LIN {X 0,Y 383.746,Z 842.553,A -85,B 0,C 180,E1 14810.521,E2 14810.521} C_VEL
LIN {X 0,Y 388.275,Z 838.57,A -85,B 0,C 180,E1 14810.091,E2 14810.091} C_VEL
LIN {X 0,Y 383.695,Z 874.566,A -85,B 0,C 180,E1 14809.08,E2 14809.08} C_VEL
LIN {X 0,Y 381.946,Z 882.091,A -85,B 0,C 180,E1 14808.965,E2 14808.965} C_VEL
LIN {X 0,Y 374.562,Z 902.014,A -85,B 0,C 180,E1 14808.987,E2 14808.987} C_VEL
LIN {X 0,Y 373.141,Z 908.472,A -85,B 0,C 180,E1 14808.863,E2 14808.863} C_VEL
LIN {X 0,Y 363.178,Z 988.067,A -85,B 0,C 180,E1 14806.33,E2 14806.33} C_VEL
LIN {X 0,Y 360.037,Z 1012.069,A -85,B 0,C 180,E1 14805.364,E2 14805.364} C_VEL
LIN {X 0,Y 356.378,Z 1034.28,A -85,B 0,C 180,E1 14804.205,E2 14804.205} C_VEL
LIN {X 0,Y 351.773,Z 1057.589,A -85,B 0,C 180,E1 14802.682,E2 14802.682} C_VEL
LIN {X 0,Y 346.903,Z 1079.031,A -85,B 0,C 180,E1 14800.957,E2 14800.957} C_VEL
LIN {X 0,Y 341.537,Z 1100.164,A -85,B 0,C 180,E1 14798.901,E2 14798.901} C_VEL
LIN {X 0,Y 335.908,Z 1120.268,A -85,B 0,C 180,E1 14796.537,E2 14796.537} C_VEL
LIN {X 0,Y 330.579,Z 1138.155,A -85,B 0,C 180,E1 14794.026,E2 14794.026} C_VEL
LIN {X 0,Y 325.16,Z 1155.707,A -85,B 0,C 180,E1 14791.105,E2 14791.105} C_VEL
LIN {X 0,Y 320.4,Z 1170.927,A -85,B 0,C 180,E1 14788.115,E2 14788.115} C_VEL
LIN {X 0,Y 315.886,Z 1185.531,A -85,B 0,C 180,E1 14784.698,E2 14784.698} C_VEL
LIN {X 0,Y 312.205,Z 1197.976,A -85,B 0,C 180,E1 14781.217,E2 14781.217} C_VEL
LIN {X 0,Y 309.066,Z 1209.644,A -85,B 0,C 180,E1 14777.316,E2 14777.316} C_VEL
LIN {X 0,Y 306.838,Z 1219.359,A -85,B 0,C 180,E1 14773.378,E2 14773.378} C_VEL
LIN {X 0,Y 305.434,Z 1227.199,A -85,B 0,C 180,E1 14769.421,E2 14769.421} C_VEL
LIN {X 0,Y 304.675,Z 1233.378,A -85,B 0,C 180,E1 14765.461,E2 14765.461} C_VEL
LIN {X 0,Y 304.399,Z 1238.104,A -85,B 0,C 180,E1 14761.506,E2 14761.506} C_VEL
LIN {X 0,Y 304.384,Z 1241.144,A -85,B 0,C 180,E1 14757.741,E2 14757.741} C_VEL
LIN {X 0,Y 304.604,Z 1243.124,A -85,B 0,C 180,E1 14753.781,E2 14753.781} C_VEL
LIN {X 0,Y 305.158,Z 1243.715,A -85,B 0,C 180,E1 14749.808,E2 14749.808} C_VEL
LIN {X 0,Y 306.521,Z 1242.868,A -85,B 0,C 180,E1 14745.26,E2 14745.26} C_VEL
LIN {X 0,Y 309.14,Z 1240.272,A -85,B 0,C 180,E1 14740.54,E2 14740.54} C_VEL
LIN {X 0,Y 313.102,Z 1236.128,A -85,B 0,C 180,E1 14736.073,E2 14736.073} C_VEL
LIN {X 0,Y 318.886,Z 1230.051,A -85,B 0,C 180,E1 14731.536,E2 14731.536} C_VEL
LIN {X 0,Y 326.471,Z 1222.117,A -85,B 0,C 180,E1 14727.173,E2 14727.173} C_VEL
LIN {X 0,Y 335.463,Z 1212.699,A -85,B 0,C 180,E1 14723.194,E2 14723.194} C_VEL
LIN {X 0,Y 346.318,Z 1201.267,A -85,B 0,C 180,E1 14719.408,E2 14719.408} C_VEL
LIN {X 0,Y 359.067,Z 1187.767,A -85,B 0,C 180,E1 14715.879,E2 14715.879} C_VEL
LIN {X 0,Y 366.745,Z 1179.688,A -85,B 0,C 180,E1 14714.081,E2 14714.081} C_VEL
LIN {X 0,Y 351.897,Z 1193.932,A -85,B 0,C 180,E1 14711.242,E2 14711.242} C_VEL
LIN {X 0,Y 336.916,Z 1211.003,A -85,B 0,C 180,E1 14707.262,E2 14707.262} C_VEL
LIN {X 0,Y 323.989,Z 1229.125,A -85,B 0,C 180,E1 14702.262,E2 14702.262} C_VEL
LIN {X 0,Y 315.462,Z 1243.813,A -85,B 0,C 180,E1 14697.363,E2 14697.363} C_VEL
LIN {X 0,Y 310.275,Z 1254.664,A -85,B 0,C 180,E1 14692.953,E2 14692.953} C_VEL
LIN {X 0,Y 306.948,Z 1263.193,A -85,B 0,C 180,E1 14688.619,E2 14688.619} C_VEL
LIN {X 0,Y 305.097,Z 1269.475,A -85,B 0,C 180,E1 14684.425,E2 14684.425} C_VEL
LIN {X 0,Y 304.326,Z 1273.688,A -85,B 0,C 180,E1 14680.413,E2 14680.413} C_VEL
LIN {X 0,Y 304.222,Z 1276.03,A -85,B 0,C 180,E1 14676.608,E2 14676.608} C_VEL
LIN {X 0,Y 304.399,Z 1276.705,A -85,B 0,C 180,E1 14673.015,E2 14673.015} C_VEL
LIN {X 0,Y 304.56,Z 1275.912,A -85,B 0,C 180,E1 14669.626,E2 14669.626} C_VEL
LIN {X 0,Y 304.568,Z 1273.68,A -85,B 0,C 180,E1 14666.238,E2 14666.238} C_VEL
LIN {X 0,Y 304.521,Z 1269.98,A -85,B 0,C 180,E1 14662.835,E2 14662.835} C_VEL
LIN {X 0,Y 304.622,Z 1264.454,A -85,B 0,C 180,E1 14659.219,E2 14659.219} C_VEL
LIN {X 0,Y 305.152,Z 1256.818,A -85,B 0,C 180,E1 14655.389,E2 14655.389} C_VEL
LIN {X 0,Y 306.321,Z 1247.288,A -85,B 0,C 180,E1 14651.544,E2 14651.544} C_VEL
LIN {X 0,Y 308.437,Z 1235.038,A -85,B 0,C 180,E1 14647.512,E2 14647.512} C_VEL
LIN {X 0,Y 311.408,Z 1221.22,A -85,B 0,C 180,E1 14643.701,E2 14643.701} C_VEL
LIN {X 0,Y 315.633,Z 1204.223,A -85,B 0,C 180,E1 14639.759,E2 14639.759} C_VEL
LIN {X 0,Y 320.988,Z 1184.662,A -85,B 0,C 180,E1 14635.956,E2 14635.956} C_VEL
LIN {X 0,Y 327.072,Z 1163.735,A -85,B 0,C 180,E1 14632.533,E2 14632.533} C_VEL
LIN {X 0,Y 333.784,Z 1141.453,A -85,B 0,C 180,E1 14629.458,E2 14629.458} C_VEL
LIN {X 0,Y 340.841,Z 1118.152,A -85,B 0,C 180,E1 14626.745,E2 14626.745} C_VEL
LIN {X 0,Y 348.53,Z 1092.821,A -85,B 0,C 180,E1 14624.258,E2 14624.258} C_VEL
LIN {X 0,Y 356.345,Z 1066.796,A -85,B 0,C 180,E1 14622.116,E2 14622.116} C_VEL
LIN {X 0,Y 363.648,Z 1041.389,A -85,B 0,C 180,E1 14620.395,E2 14620.395} C_VEL
LIN {X 0,Y 371.162,Z 1013.758,A -85,B 0,C 180,E1 14618.876,E2 14618.876} C_VEL
LIN {X 0,Y 377.143,Z 988.406,A -85,B 0,C 180,E1 14617.706,E2 14617.706} C_VEL
LIN {X 0,Y 371.129,Z 963.994,A -85,B 0,C 180,E1 14615.41,E2 14615.41} C_VEL
LIN {X 0,Y 366.924,Z 941.456,A -85,B 0,C 180,E1 14613.531,E2 14613.531} C_VEL
LIN {X 0,Y 363.372,Z 914.987,A -85,B 0,C 180,E1 14611.591,E2 14611.591} C_VEL
LIN {X 0,Y 361.819,Z 891.552,A -85,B 0,C 180,E1 14610.013,E2 14610.013} C_VEL
LIN {X 0,Y 372.049,Z 851.191,A -85,B 0,C 180,E1 14605.212,E2 14605.212} C_VEL
LIN {X 0,Y 380.821,Z 818.494,A -85,B 0,C 180,E1 14601.324,E2 14601.324} C_VEL
LIN {X 0,Y 381.9,Z 814.099,A -85,B 0,C 180,E1 14600.787,E2 14600.787} C_VEL
LIN {X 0,Y 375.953,Z 797.311,A -85,B 0,C 180,E1 14597.011,E2 14597.011} C_VEL
LIN {X 0,Y 370.417,Z 782.695,A -85,B 0,C 180,E1 14593.423,E2 14593.423} C_VEL
LIN {X 0,Y 364.786,Z 768.438,A -85,B 0,C 180,E1 14589.625,E2 14589.625} C_VEL
LIN {X 0,Y 359.48,Z 755.657,A -85,B 0,C 180,E1 14585.907,E2 14585.907} C_VEL
LIN {X 0,Y 354.12,Z 743.204,A -85,B 0,C 180,E1 14581.942,E2 14581.942} C_VEL
LIN {X 0,Y 349.074,Z 731.964,A -85,B 0,C 180,E1 14578.03,E2 14578.03} C_VEL
LIN {X 0,Y 344.556,Z 722.244,A -85,B 0,C 180,E1 14574.338,E2 14574.338} C_VEL
LIN {X 0,Y 340.097,Z 712.564,A -85,B 0,C 180,E1 14570.353,E2 14570.353} C_VEL
LIN {X 0,Y 336.736,Z 705.94,A -85,B 0,C 180,E1 14567.307,E2 14567.307} C_VEL
LIN {X 0,Y 334.521,Z 701.406,A -85,B 0,C 180,E1 14565.104,E2 14565.104} C_VEL
LIN {X 0,Y 332.667,Z 697.681,A -85,B 0,C 180,E1 14563.229,E2 14563.229} C_VEL
LIN {X 0,Y 330.716,Z 693.689,A -85,B 0,C 180,E1 14561.125,E2 14561.125} C_VEL
LIN {X 0,Y 328.472,Z 689.184,A -85,B 0,C 180,E1 14558.575,E2 14558.575} C_VEL
LIN {X 0,Y 326.1,Z 684.518,A -85,B 0,C 180,E1 14555.74,E2 14555.74} C_VEL
LIN {X 0,Y 323.782,Z 679.957,A -85,B 0,C 180,E1 14552.79,E2 14552.79} C_VEL
LIN {X 0,Y 321.463,Z 675.343,A -85,B 0,C 180,E1 14549.535,E2 14549.535} C_VEL
LIN {X 0,Y 323.347,Z 676.36,A -85,B 0,C 180,E1 14548.908,E2 14548.908} C_VEL
LIN {X 0,Y 329.514,Z 688.003,A -85,B 0,C 180,E1 14545.849,E2 14545.849} C_VEL
LIN {X 0,Y 335.679,Z 701.279,A -85,B 0,C 180,E1 14542.794,E2 14542.794} C_VEL
LIN {X 0,Y 341.917,Z 716.478,A -85,B 0,C 180,E1 14539.738,E2 14539.738} C_VEL
LIN {X 0,Y 347.429,Z 732.534,A -85,B 0,C 180,E1 14536.88,E2 14536.88} C_VEL
LIN {X 0,Y 352.001,Z 748.58,A -85,B 0,C 180,E1 14534.341,E2 14534.341} C_VEL
LIN {X 0,Y 346.421,Z 794.632,A -85,B 0,C 180,E1 14530.169,E2 14530.169} C_VEL
LIN {X 0,Y 340.819,Z 844.347,A -85,B 0,C 180,E1 14525.716,E2 14525.716} C_VEL
LIN {X 0,Y 338.058,Z 873.297,A -85,B 0,C 180,E1 14523.219,E2 14523.219} C_VEL
LIN {X 0,Y 338.378,Z 880.004,A -85,B 0,C 180,E1 14523.012,E2 14523.012} C_VEL
LIN {X 0,Y 332.419,Z 1032.548,A -85,B 0,C 180,E1 14519.855,E2 14519.855} C_VEL
LIN {X 0,Y 331.822,Z 1052.049,A -85,B 0,C 180,E1 14519.278,E2 14519.278} C_VEL
LIN {X 0,Y 330.671,Z 1068.771,A -85,B 0,C 180,E1 14518.487,E2 14518.487} C_VEL
LIN {X 0,Y 328.942,Z 1084.738,A -85,B 0,C 180,E1 14517.426,E2 14517.426} C_VEL
LIN {X 0,Y 326.673,Z 1100.489,A -85,B 0,C 180,E1 14516.052,E2 14516.052} C_VEL
LIN {X 0,Y 324.079,Z 1115.176,A -85,B 0,C 180,E1 14514.418,E2 14514.418} C_VEL
LIN {X 0,Y 321.235,Z 1128.864,A -85,B 0,C 180,E1 14512.508,E2 14512.508} C_VEL
LIN {X 0,Y 318.391,Z 1140.966,A -85,B 0,C 180,E1 14510.398,E2 14510.398} C_VEL
LIN {X 0,Y 315.444,Z 1152.469,A -85,B 0,C 180,E1 14507.904,E2 14507.904} C_VEL
LIN {X 0,Y 312.77,Z 1162.396,A -85,B 0,C 180,E1 14505.195,E2 14505.195} C_VEL
LIN {X 0,Y 310.464,Z 1170.688,A -85,B 0,C 180,E1 14502.27,E2 14502.27} C_VEL
LIN {X 0,Y 308.629,Z 1177.374,A -85,B 0,C 180,E1 14499.132,E2 14499.132} C_VEL
LIN {X 0,Y 307.388,Z 1182.154,A -85,B 0,C 180,E1 14495.972,E2 14495.972} C_VEL
LIN {X 0,Y 306.666,Z 1185.162,A -85,B 0,C 180,E1 14492.801,E2 14492.801} C_VEL
LIN {X 0,Y 306.392,Z 1186.519,A -85,B 0,C 180,E1 14489.437,E2 14489.437} C_VEL
LIN {X 0,Y 306.581,Z 1186.104,A -85,B 0,C 180,E1 14486.07,E2 14486.07} C_VEL
LIN {X 0,Y 307.219,Z 1184.055,A -85,B 0,C 180,E1 14482.893,E2 14482.893} C_VEL
LIN {X 0,Y 308.37,Z 1180.265,A -85,B 0,C 180,E1 14479.725,E2 14479.725} C_VEL
LIN {X 0,Y 310.095,Z 1174.632,A -85,B 0,C 180,E1 14476.573,E2 14476.573} C_VEL
LIN {X 0,Y 312.31,Z 1167.487,A -85,B 0,C 180,E1 14473.634,E2 14473.634} C_VEL
LIN {X 0,Y 314.919,Z 1158.895,A -85,B 0,C 180,E1 14470.909,E2 14470.909} C_VEL
LIN {X 0,Y 317.812,Z 1148.821,A -85,B 0,C 180,E1 14468.399,E2 14468.399} C_VEL
LIN {X 0,Y 320.876,Z 1137.312,A -85,B 0,C 180,E1 14466.101,E2 14466.101} C_VEL
LIN {X 0,Y 324.011,Z 1124.278,A -85,B 0,C 180,E1 14464.008,E2 14464.008} C_VEL
LIN {X 0,Y 326.967,Z 1110.208,A -85,B 0,C 180,E1 14462.2,E2 14462.2} C_VEL
LIN {X 0,Y 329.607,Z 1094.995,A -85,B 0,C 180,E1 14460.662,E2 14460.662} C_VEL
LIN {X 0,Y 331.831,Z 1078.659,A -85,B 0,C 180,E1 14459.385,E2 14459.385} C_VEL
LIN {X 0,Y 333.495,Z 1061.599,A -85,B 0,C 180,E1 14458.396,E2 14458.396} C_VEL
LIN {X 0,Y 334.442,Z 1044.124,A -85,B 0,C 180,E1 14457.715,E2 14457.715} C_VEL
LIN {X 0,Y 335.857,Z 997.984,A -85,B 0,C 180,E1 14456.674,E2 14456.674} C_VEL
LIN {X 0,Y 340.682,Z 888.138,A -85,B 0,C 180,E1 14454.417,E2 14454.417} C_VEL
LIN {X 0,Y 342.316,Z 888.44,A -85,B 0,C 180,E1 14454.149,E2 14454.149} C_VEL
LIN {X 0,Y 344.514,Z 886.501,A -85,B 0,C 180,E1 14453.925,E2 14453.925} C_VEL
LIN {X 0,Y 347.947,Z 880.496,A -85,B 0,C 180,E1 14453.739,E2 14453.739} C_VEL
LIN {X 0,Y 349.926,Z 876.513,A -85,B 0,C 180,E1 14453.661,E2 14453.661} C_VEL
LIN {X 0,Y 354.255,Z 874.098,A -85,B 0,C 180,E1 14453.143,E2 14453.143} C_VEL
LIN {X 0,Y 358.913,Z 869.497,A -85,B 0,C 180,E1 14452.702,E2 14452.702} C_VEL
LIN {X 0,Y 365.117,Z 865.492,A -85,B 0,C 180,E1 14452.011,E2 14452.011} C_VEL
LIN {X 0,Y 369.888,Z 861.076,A -85,B 0,C 180,E1 14451.555,E2 14451.555} C_VEL
LIN {X 0,Y 375.918,Z 856.95,A -85,B 0,C 180,E1 14450.919,E2 14450.919} C_VEL
LIN {X 0,Y 380.175,Z 853.157,A -85,B 0,C 180,E1 14450.517,E2 14450.517} C_VEL
LIN {X 0,Y 380.46,Z 853.179,A -85,B 0,C 180,E1 14450.477,E2 14450.477} C_VEL
LIN {X 0,Y 373.141,Z 908.472,A -85,B 0,C 180,E1 14448.863,E2 14448.863} C_VEL
LIN {X 0,Y 371.361,Z 915.986,A -85,B 0,C 180,E1 14448.736,E2 14448.736} C_VEL
LIN {X 0,Y 363.787,Z 935.843,A -85,B 0,C 180,E1 14448.725,E2 14448.725} C_VEL
LIN {X 0,Y 362.352,Z 942.286,A -85,B 0,C 180,E1 14448.588,E2 14448.588} C_VEL
LIN {X 0,Y 355.036,Z 1000.064,A -85,B 0,C 180,E1 14446.594,E2 14446.594} C_VEL
LIN {X 0,Y 351.627,Z 1022.777,A -85,B 0,C 180,E1 14445.541,E2 14445.541} C_VEL
LIN {X 0,Y 347.34,Z 1046.129,A -85,B 0,C 180,E1 14444.159,E2 14444.159} C_VEL
LIN {X 0,Y 342.711,Z 1067.461,A -85,B 0,C 180,E1 14442.601,E2 14442.601} C_VEL
LIN {X 0,Y 337.432,Z 1088.949,A -85,B 0,C 180,E1 14440.686,E2 14440.686} C_VEL
LIN {X 0,Y 331.833,Z 1109.386,A -85,B 0,C 180,E1 14438.48,E2 14438.48} C_VEL
LIN {X 0,Y 326.28,Z 1128.261,A -85,B 0,C 180,E1 14436.043,E2 14436.043} C_VEL
LIN {X 0,Y 320.49,Z 1146.894,A -85,B 0,C 180,E1 14433.176,E2 14433.176} C_VEL
LIN {X 0,Y 315.42,Z 1162.839,A -85,B 0,C 180,E1 14430.268,E2 14430.268} C_VEL
LIN {X 0,Y 310.338,Z 1178.724,A -85,B 0,C 180,E1 14426.81,E2 14426.81} C_VEL
LIN {X 0,Y 306.13,Z 1192.235,A -85,B 0,C 180,E1 14423.279,E2 14423.279} C_VEL
LIN {X 0,Y 302.608,Z 1204.374,A -85,B 0,C 180,E1 14419.495,E2 14419.495} C_VEL
LIN {X 0,Y 299.977,Z 1214.644,A -85,B 0,C 180,E1 14415.664,E2 14415.664} C_VEL
LIN {X 0,Y 298.104,Z 1223.506,A -85,B 0,C 180,E1 14411.61,E2 14411.61} C_VEL
LIN {X 0,Y 296.995,Z 1230.615,A -85,B 0,C 180,E1 14407.545,E2 14407.545} C_VEL
LIN {X 0,Y 296.494,Z 1236.194,A -85,B 0,C 180,E1 14403.48,E2 14403.48} C_VEL
LIN {X 0,Y 296.374,Z 1240.036,A -85,B 0,C 180,E1 14399.613,E2 14399.613} C_VEL
LIN {X 0,Y 296.488,Z 1242.863,A -85,B 0,C 180,E1 14395.357,E2 14395.357} C_VEL
LIN {X 0,Y 296.921,Z 1244.215,A -85,B 0,C 180,E1 14391.284,E2 14391.284} C_VEL
LIN {X 0,Y 297.971,Z 1244.194,A -85,B 0,C 180,E1 14386.81,E2 14386.81} C_VEL
LIN {X 0,Y 300.24,Z 1242.517,A -85,B 0,C 180,E1 14381.958,E2 14381.958} C_VEL
LIN {X 0,Y 304.013,Z 1239.12,A -85,B 0,C 180,E1 14377.164,E2 14377.164} C_VEL
LIN {X 0,Y 309.508,Z 1233.987,A -85,B 0,C 180,E1 14372.485,E2 14372.485} C_VEL
LIN {X 0,Y 316.836,Z 1227.095,A -85,B 0,C 180,E1 14367.982,E2 14367.982} C_VEL
LIN {X 0,Y 326.049,Z 1218.391,A -85,B 0,C 180,E1 14363.71,E2 14363.71} C_VEL
LIN {X 0,Y 337.135,Z 1207.821,A -85,B 0,C 180,E1 14359.717,E2 14359.717} C_VEL
LIN {X 0,Y 350.229,Z 1195.277,A -85,B 0,C 180,E1 14356.011,E2 14356.011} C_VEL
LIN {X 0,Y 357.971,Z 1187.89,A -85,B 0,C 180,E1 14354.182,E2 14354.182} C_VEL
LIN {X 0,Y 342.431,Z 1202.026,A -85,B 0,C 180,E1 14351.073,E2 14351.073} C_VEL
LIN {X 0,Y 327.659,Z 1217.995,A -85,B 0,C 180,E1 14346.956,E2 14346.956} C_VEL
LIN {X 0,Y 314.933,Z 1234.715,A -85,B 0,C 180,E1 14341.808,E2 14341.808} C_VEL
LIN {X 0,Y 306.554,Z 1248.183,A -85,B 0,C 180,E1 14336.754,E2 14336.754} C_VEL
LIN {X 0,Y 301.384,Z 1258.338,A -85,B 0,C 180,E1 14332.02,E2 14332.02} C_VEL
LIN {X 0,Y 298.359,Z 1265.813,A -85,B 0,C 180,E1 14327.557,E2 14327.557} C_VEL
LIN {X 0,Y 296.743,Z 1271.328,A -85,B 0,C 180,E1 14323.05,E2 14323.05} C_VEL
LIN {X 0,Y 296.226,Z 1274.562,A -85,B 0,C 180,E1 14318.935,E2 14318.935} C_VEL
LIN {X 0,Y 296.294,Z 1275.941,A -85,B 0,C 180,E1 14315.23,E2 14315.23} C_VEL
LIN {X 0,Y 296.515,Z 1275.809,A -85,B 0,C 180,E1 14311.548,E2 14311.548} C_VEL
LIN {X 0,Y 296.621,Z 1274.367,A -85,B 0,C 180,E1 14308.264,E2 14308.264} C_VEL
LIN {X 0,Y 296.59,Z 1271.419,A -85,B 0,C 180,E1 14304.78,E2 14304.78} C_VEL
LIN {X 0,Y 296.565,Z 1266.986,A -85,B 0,C 180,E1 14301.276,E2 14301.276} C_VEL
LIN {X 0,Y 296.821,Z 1260.651,A -85,B 0,C 180,E1 14297.552,E2 14297.552} C_VEL
LIN {X 0,Y 297.622,Z 1252.148,A -85,B 0,C 180,E1 14293.611,E2 14293.611} C_VEL
LIN {X 0,Y 299.172,Z 1241.673,A -85,B 0,C 180,E1 14289.663,E2 14289.663} C_VEL
LIN {X 0,Y 301.778,Z 1228.416,A -85,B 0,C 180,E1 14285.536,E2 14285.536} C_VEL
LIN {X 0,Y 305.101,Z 1214.292,A -85,B 0,C 180,E1 14281.834,E2 14281.834} C_VEL
LIN {X 0,Y 309.645,Z 1197.173,A -85,B 0,C 180,E1 14278.026,E2 14278.026} C_VEL
LIN {X 0,Y 315.287,Z 1177.61,A -85,B 0,C 180,E1 14274.362,E2 14274.362} C_VEL
LIN {X 0,Y 321.53,Z 1156.956,A -85,B 0,C 180,E1 14271.088,E2 14271.088} C_VEL
LIN {X 0,Y 328.465,Z 1134.516,A -85,B 0,C 180,E1 14268.077,E2 14268.077} C_VEL
LIN {X 0,Y 336.889,Z 1107.478,A -85,B 0,C 180,E1 14265.063,E2 14265.063} C_VEL
LIN {X 0,Y 344.781,Z 1082.032,A -85,B 0,C 180,E1 14262.683,E2 14262.683} C_VEL
LIN {X 0,Y 352.629,Z 1056.096,A -85,B 0,C 180,E1 14260.684,E2 14260.684} C_VEL
LIN {X 0,Y 360.592,Z 1028.573,A -85,B 0,C 180,E1 14258.945,E2 14258.945} C_VEL
LIN {X 0,Y 367.813,Z 1001.505,A -85,B 0,C 180,E1 14257.549,E2 14257.549} C_VEL
LIN {X 0,Y 370.29,Z 990.176,A -85,B 0,C 180,E1 14257.025,E2 14257.025} C_VEL
LIN {X 0,Y 364.693,Z 965.814,A -85,B 0,C 180,E1 14254.667,E2 14254.667} C_VEL
LIN {X 0,Y 360.301,Z 940.519,A -85,B 0,C 180,E1 14252.535,E2 14252.535} C_VEL
LIN {X 0,Y 357.231,Z 914.188,A -85,B 0,C 180,E1 14250.59,E2 14250.59} C_VEL
LIN {X 0,Y 355.891,Z 889.583,A -85,B 0,C 180,E1 14248.941,E2 14248.941} C_VEL
LIN {X 0,Y 365.743,Z 852.148,A -85,B 0,C 180,E1 14244.45,E2 14244.45} C_VEL
LIN {X 0,Y 374.483,Z 820.314,A -85,B 0,C 180,E1 14240.637,E2 14240.637} C_VEL
LIN {X 0,Y 375.145,Z 817.467,A -85,B 0,C 180,E1 14240.273,E2 14240.273} C_VEL
LIN {X 0,Y 369.598,Z 801.679,A -85,B 0,C 180,E1 14236.665,E2 14236.665} C_VEL
LIN {X 0,Y 364.088,Z 787.029,A -85,B 0,C 180,E1 14233.014,E2 14233.014} C_VEL
LIN {X 0,Y 358.292,Z 772.182,A -85,B 0,C 180,E1 14228.991,E2 14228.991} C_VEL
LIN {X 0,Y 352.77,Z 758.933,A -85,B 0,C 180,E1 14225.041,E2 14225.041} C_VEL
LIN {X 0,Y 347.641,Z 746.903,A -85,B 0,C 180,E1 14221.154,E2 14221.154} C_VEL
LIN {X 0,Y 342.056,Z 734.282,A -85,B 0,C 180,E1 14216.648,E2 14216.648} C_VEL
LIN {X 0,Y 336.652,Z 722.607,A -85,B 0,C 180,E1 14211.976,E2 14211.976} C_VEL
LIN {X 0,Y 332.172,Z 713.221,A -85,B 0,C 180,E1 14207.836,E2 14207.836} C_VEL
LIN {X 0,Y 328.212,Z 704.901,A -85,B 0,C 180,E1 14203.814,E2 14203.814} C_VEL
LIN {X 0,Y 325.086,Z 699.043,A -85,B 0,C 180,E1 14200.599,E2 14200.599} C_VEL
LIN {X 0,Y 323.236,Z 695.16,A -85,B 0,C 180,E1 14198.401,E2 14198.401} C_VEL
LIN {X 0,Y 320.841,Z 690.451,A -85,B 0,C 180,E1 14195.499,E2 14195.499} C_VEL
LIN {X 0,Y 318.575,Z 685.943,A -85,B 0,C 180,E1 14192.524,E2 14192.524} C_VEL
LIN {X 0,Y 316.716,Z 682.164,A -85,B 0,C 180,E1 14189.869,E2 14189.869} C_VEL
LIN {X 0,Y 319.085,Z 683.348,A -85,B 0,C 180,E1 14189.075,E2 14189.075} C_VEL
LIN {X 0,Y 324.101,Z 693.003,A -85,B 0,C 180,E1 14186.479,E2 14186.479} C_VEL
LIN {X 0,Y 330.142,Z 706.097,A -85,B 0,C 180,E1 14183.37,E2 14183.37} C_VEL
LIN {X 0,Y 336.189,Z 721.204,A -85,B 0,C 180,E1 14180.249,E2 14180.249} C_VEL
LIN {X 0,Y 341.489,Z 736.768,A -85,B 0,C 180,E1 14177.439,E2 14177.439} C_VEL
LIN {X 0,Y 345.719,Z 751.902,A -85,B 0,C 180,E1 14174.997,E2 14174.997} C_VEL
LIN {X 0,Y 339.578,Z 800.369,A -85,B 0,C 180,E1 14170.563,E2 14170.563} C_VEL
LIN {X 0,Y 333.79,Z 850.487,A -85,B 0,C 180,E1 14166.046,E2 14166.046} C_VEL
LIN {X 0,Y 331.464,Z 874.294,A -85,B 0,C 180,E1 14163.981,E2 14163.981} C_VEL
LIN {X 0,Y 331.759,Z 880.873,A -85,B 0,C 180,E1 14163.774,E2 14163.774} C_VEL
LIN {X 0,Y 325.585,Z 1032.92,A -85,B 0,C 180,E1 14160.577,E2 14160.577} C_VEL
LIN {X 0,Y 324.956,Z 1052.733,A -85,B 0,C 180,E1 14159.985,E2 14159.985} C_VEL
LIN {X 0,Y 323.721,Z 1069.933,A -85,B 0,C 180,E1 14159.157,E2 14159.157} C_VEL
LIN {X 0,Y 321.925,Z 1085.838,A -85,B 0,C 180,E1 14158.077,E2 14158.077} C_VEL
LIN {X 0,Y 319.567,Z 1101.568,A -85,B 0,C 180,E1 14156.676,E2 14156.676} C_VEL
LIN {X 0,Y 316.874,Z 1116.233,A -85,B 0,C 180,E1 14155.011,E2 14155.011} C_VEL
LIN {X 0,Y 313.921,Z 1129.897,A -85,B 0,C 180,E1 14153.062,E2 14153.062} C_VEL
LIN {X 0,Y 310.966,Z 1141.986,A -85,B 0,C 180,E1 14150.908,E2 14150.908} C_VEL
LIN {X 0,Y 307.901,Z 1153.479,A -85,B 0,C 180,E1 14148.358,E2 14148.358} C_VEL
LIN {X 0,Y 305.115,Z 1163.396,A -85,B 0,C 180,E1 14145.585,E2 14145.585} C_VEL
LIN {X 0,Y 302.708,Z 1171.676,A -85,B 0,C 180,E1 14142.589,E2 14142.589} C_VEL
LIN {X 0,Y 300.79,Z 1178.355,A -85,B 0,C 180,E1 14139.372,E2 14139.372} C_VEL
LIN {X 0,Y 299.49,Z 1183.126,A -85,B 0,C 180,E1 14136.13,E2 14136.13} C_VEL
LIN {X 0,Y 298.733,Z 1186.124,A -85,B 0,C 180,E1 14132.875,E2 14132.875} C_VEL
LIN {X 0,Y 298.448,Z 1187.473,A -85,B 0,C 180,E1 14129.422,E2 14129.422} C_VEL
LIN {X 0,Y 298.651,Z 1187.052,A -85,B 0,C 180,E1 14125.966,E2 14125.966} C_VEL
LIN {X 0,Y 299.327,Z 1184.996,A -85,B 0,C 180,E1 14122.705,E2 14122.705} C_VEL
LIN {X 0,Y 300.54,Z 1181.195,A -85,B 0,C 180,E1 14119.454,E2 14119.454} C_VEL
LIN {X 0,Y 302.355,Z 1175.554,A -85,B 0,C 180,E1 14116.223,E2 14116.223} C_VEL
LIN {X 0,Y 304.677,Z 1168.399,A -85,B 0,C 180,E1 14113.212,E2 14113.212} C_VEL
LIN {X 0,Y 307.405,Z 1159.794,A -85,B 0,C 180,E1 14110.424,E2 14110.424} C_VEL
LIN {X 0,Y 310.423,Z 1149.704,A -85,B 0,C 180,E1 14107.858,E2 14107.858} C_VEL
LIN {X 0,Y 313.614,Z 1138.179,A -85,B 0,C 180,E1 14105.511,E2 14105.511} C_VEL
LIN {X 0,Y 316.876,Z 1125.128,A -85,B 0,C 180,E1 14103.377,E2 14103.377} C_VEL
LIN {X 0,Y 319.947,Z 1111.023,A -85,B 0,C 180,E1 14101.535,E2 14101.535} C_VEL
LIN {X 0,Y 322.689,Z 1095.774,A -85,B 0,C 180,E1 14099.969,E2 14099.969} C_VEL
LIN {X 0,Y 325.001,Z 1079.387,A -85,B 0,C 180,E1 14098.669,E2 14098.669} C_VEL
LIN {X 0,Y 326.722,Z 1062.309,A -85,B 0,C 180,E1 14097.667,E2 14097.667} C_VEL
LIN {X 0,Y 327.702,Z 1044.822,A -85,B 0,C 180,E1 14096.979,E2 14096.979} C_VEL
LIN {X 0,Y 329.198,Z 998.297,A -85,B 0,C 180,E1 14095.912,E2 14095.912} C_VEL
LIN {X 0,Y 333.023,Z 912.972,A -85,B 0,C 180,E1 14094.134,E2 14094.134} C_VEL
LIN {X 0,Y 334.348,Z 913.487,A -85,B 0,C 180,E1 14093.902,E2 14093.902} C_VEL
LIN {X 0,Y 336.432,Z 912.104,A -85,B 0,C 180,E1 14093.668,E2 14093.668} C_VEL
LIN {X 0,Y 339.643,Z 907.293,A -85,B 0,C 180,E1 14093.47,E2 14093.47} C_VEL
LIN {X 0,Y 343.59,Z 897.918,A -85,B 0,C 180,E1 14093.419,E2 14093.419} C_VEL
LIN {X 0,Y 344.782,Z 894.808,A -85,B 0,C 180,E1 14093.416,E2 14093.416} C_VEL
LIN {X 0,Y 348.332,Z 891.335,A -85,B 0,C 180,E1 14093.081,E2 14093.081} C_VEL
LIN {X 0,Y 352.21,Z 884.946,A -85,B 0,C 180,E1 14092.86,E2 14092.86} C_VEL
LIN {X 0,Y 353.522,Z 882.532,A -85,B 0,C 180,E1 14092.8,E2 14092.8} C_VEL
LIN {X 0,Y 358.945,Z 878.474,A -85,B 0,C 180,E1 14092.228,E2 14092.228} C_VEL
LIN {X 0,Y 362.079,Z 875.507,A -85,B 0,C 180,E1 14091.936,E2 14091.936} C_VEL
LIN {X 0,Y 367.945,Z 871.521,A -85,B 0,C 180,E1 14091.314,E2 14091.314} C_VEL
LIN {X 0,Y 372.549,Z 867.452,A -85,B 0,C 180,E1 14090.878,E2 14090.878} C_VEL
LIN {X 0,Y 362.352,Z 942.286,A -85,B 0,C 180,E1 14088.588,E2 14088.588} C_VEL
LIN {X 0,Y 360.573,Z 949.783,A -85,B 0,C 180,E1 14088.439,E2 14088.439} C_VEL
LIN {X 0,Y 352.922,Z 969.594,A -85,B 0,C 180,E1 14088.373,E2 14088.373} C_VEL
LIN {X 0,Y 351.459,Z 976.022,A -85,B 0,C 180,E1 14088.222,E2 14088.222} C_VEL
LIN {X 0,Y 347.325,Z 1007.823,A -85,B 0,C 180,E1 14086.989,E2 14086.989} C_VEL
LIN {X 0,Y 343.59,Z 1030.541,A -85,B 0,C 180,E1 14085.836,E2 14085.836} C_VEL
LIN {X 0,Y 338.978,Z 1053.543,A -85,B 0,C 180,E1 14084.354,E2 14084.354} C_VEL
LIN {X 0,Y 334.066,Z 1074.568,A -85,B 0,C 180,E1 14082.683,E2 14082.683} C_VEL
LIN {X 0,Y 328.541,Z 1095.781,A -85,B 0,C 180,E1 14080.639,E2 14080.639} C_VEL
LIN {X 0,Y 322.74,Z 1116.035,A -85,B 0,C 180,E1 14078.289,E2 14078.289} C_VEL
LIN {X 0,Y 316.999,Z 1134.723,A -85,B 0,C 180,E1 14075.7,E2 14075.7} C_VEL
LIN {X 0,Y 311.155,Z 1152.906,A -85,B 0,C 180,E1 14072.675,E2 14072.675} C_VEL
LIN {X 0,Y 305.714,Z 1169.421,A -85,B 0,C 180,E1 14069.38,E2 14069.38} C_VEL
LIN {X 0,Y 301.079,Z 1183.668,A -85,B 0,C 180,E1 14066,E2 14066} C_VEL
LIN {X 0,Y 297.038,Z 1196.636,A -85,B 0,C 180,E1 14062.357,E2 14062.357} C_VEL
LIN {X 0,Y 293.591,Z 1208.768,A -85,B 0,C 180,E1 14058.26,E2 14058.26} C_VEL
LIN {X 0,Y 291.126,Z 1218.758,A -85,B 0,C 180,E1 14054.114,E2 14054.114} C_VEL
LIN {X 0,Y 289.557,Z 1226.947,A -85,B 0,C 180,E1 14049.943,E2 14049.943} C_VEL
LIN {X 0,Y 288.716,Z 1233.519,A -85,B 0,C 180,E1 14045.764,E2 14045.764} C_VEL
LIN {X 0,Y 288.41,Z 1238.238,A -85,B 0,C 180,E1 14041.788,E2 14041.788} C_VEL
LIN {X 0,Y 288.399,Z 1241.848,A -85,B 0,C 180,E1 14037.616,E2 14037.616} C_VEL
LIN {X 0,Y 288.635,Z 1243.997,A -85,B 0,C 180,E1 14033.635,E2 14033.635} C_VEL
LIN {X 0,Y 289.361,Z 1245.037,A -85,B 0,C 180,E1 14029.044,E2 14029.044} C_VEL
LIN {X 0,Y 290.932,Z 1244.626,A -85,B 0,C 180,E1 14024.45,E2 14024.45} C_VEL
LIN {X 0,Y 293.991,Z 1242.532,A -85,B 0,C 180,E1 14019.493,E2 14019.493} C_VEL
LIN {X 0,Y 298.97,Z 1238.529,A -85,B 0,C 180,E1 14014.441,E2 14014.441} C_VEL
LIN {X 0,Y 306.266,Z 1232.437,A -85,B 0,C 180,E1 14009.382,E2 14009.382} C_VEL
LIN {X 0,Y 315.414,Z 1224.679,A -85,B 0,C 180,E1 14004.763,E2 14004.763} C_VEL
LIN {X 0,Y 326.642,Z 1215.027,A -85,B 0,C 180,E1 14000.453,E2 14000.453} C_VEL
LIN {X 0,Y 339.918,Z 1203.516,A -85,B 0,C 180,E1 13996.502,E2 13996.502} C_VEL
LIN {X 0,Y 349.008,Z 1195.671,A -85,B 0,C 180,E1 13994.269,E2 13994.269} C_VEL
LIN {X 0,Y 332.904,Z 1209.528,A -85,B 0,C 180,E1 13990.905,E2 13990.905} C_VEL
LIN {X 0,Y 317.859,Z 1224.925,A -85,B 0,C 180,E1 13986.482,E2 13986.482} C_VEL
LIN {X 0,Y 305.817,Z 1239.836,A -85,B 0,C 180,E1 13981.325,E2 13981.325} C_VEL
LIN {X 0,Y 297.891,Z 1251.707,A -85,B 0,C 180,E1 13976.302,E2 13976.302} C_VEL
LIN {X 0,Y 292.851,Z 1260.878,A -85,B 0,C 180,E1 13971.431,E2 13971.431} C_VEL
LIN {X 0,Y 289.987,Z 1267.489,A -85,B 0,C 180,E1 13966.839,E2 13966.839} C_VEL
LIN {X 0,Y 288.599,Z 1272.019,A -85,B 0,C 180,E1 13962.407,E2 13962.407} C_VEL
LIN {X 0,Y 288.221,Z 1274.612,A -85,B 0,C 180,E1 13958.18,E2 13958.18} C_VEL
LIN {X 0,Y 288.374,Z 1275.434,A -85,B 0,C 180,E1 13954.178,E2 13954.178} C_VEL
LIN {X 0,Y 288.602,Z 1274.743,A -85,B 0,C 180,E1 13950.598,E2 13950.598} C_VEL
LIN {X 0,Y 288.663,Z 1272.796,A -85,B 0,C 180,E1 13947.223,E2 13947.223} C_VEL
LIN {X 0,Y 288.611,Z 1269.275,A -85,B 0,C 180,E1 13943.638,E2 13943.638} C_VEL
LIN {X 0,Y 288.661,Z 1263.912,A -85,B 0,C 180,E1 13939.828,E2 13939.828} C_VEL
LIN {X 0,Y 289.121,Z 1256.42,A -85,B 0,C 180,E1 13935.789,E2 13935.789} C_VEL
LIN {X 0,Y 290.248,Z 1247.008,A -85,B 0,C 180,E1 13931.733,E2 13931.733} C_VEL
LIN {X 0,Y 292.247,Z 1235.573,A -85,B 0,C 180,E1 13927.684,E2 13927.684} C_VEL
LIN {X 0,Y 295.41,Z 1221.259,A -85,B 0,C 180,E1 13923.466,E2 13923.466} C_VEL
LIN {X 0,Y 299.537,Z 1205.235,A -85,B 0,C 180,E1 13919.513,E2 13919.513} C_VEL
LIN {X 0,Y 304.545,Z 1187.637,A -85,B 0,C 180,E1 13915.83,E2 13915.83} C_VEL
LIN {X 0,Y 310.953,Z 1166.56,A -85,B 0,C 180,E1 13912.112,E2 13912.112} C_VEL
LIN {X 0,Y 318.211,Z 1143.53,A -85,B 0,C 180,E1 13908.714,E2 13908.714} C_VEL
LIN {X 0,Y 325.67,Z 1120.005,A -85,B 0,C 180,E1 13905.822,E2 13905.822} C_VEL
LIN {X 0,Y 333.815,Z 1094.522,A -85,B 0,C 180,E1 13903.171,E2 13903.171} C_VEL
LIN {X 0,Y 341.747,Z 1069.36,A -85,B 0,C 180,E1 13900.991,E2 13900.991} C_VEL
LIN {X 0,Y 350.075,Z 1041.901,A -85,B 0,C 180,E1 13899.028,E2 13899.028} C_VEL
LIN {X 0,Y 357.801,Z 1015.152,A -85,B 0,C 180,E1 13897.477,E2 13897.477} C_VEL
LIN {X 0,Y 363.514,Z 992.143,A -85,B 0,C 180,E1 13896.353,E2 13896.353} C_VEL
LIN {X 0,Y 358.658,Z 970.255,A -85,B 0,C 180,E1 13894.177,E2 13894.177} C_VEL
LIN {X 0,Y 354.566,Z 945.023,A -85,B 0,C 180,E1 13891.949,E2 13891.949} C_VEL
LIN {X 0,Y 351.457,Z 917.797,A -85,B 0,C 180,E1 13889.883,E2 13889.883} C_VEL
LIN {X 0,Y 349.984,Z 890.311,A -85,B 0,C 180,E1 13888.036,E2 13888.036} C_VEL
LIN {X 0,Y 350.08,Z 887.508,A -85,B 0,C 180,E1 13887.839,E2 13887.839} C_VEL
LIN {X 0,Y 359.619,Z 852.542,A -85,B 0,C 180,E1 13883.602,E2 13883.602} C_VEL
LIN {X 0,Y 368.486,Z 821.166,A -85,B 0,C 180,E1 13879.807,E2 13879.807} C_VEL
LIN {X 0,Y 362.81,Z 804.787,A -85,B 0,C 180,E1 13875.998,E2 13875.998} C_VEL
LIN {X 0,Y 357.113,Z 789.561,A -85,B 0,C 180,E1 13872.122,E2 13872.122} C_VEL
LIN {X 0,Y 351.303,Z 774.761,A -85,B 0,C 180,E1 13868.017,E2 13868.017} C_VEL
LIN {X 0,Y 346.063,Z 762.04,A -85,B 0,C 180,E1 13864.142,E2 13864.142} C_VEL
LIN {X 0,Y 340.94,Z 750.143,A -85,B 0,C 180,E1 13860.168,E2 13860.168} C_VEL
LIN {X 0,Y 336.016,Z 738.99,A -85,B 0,C 180,E1 13856.075,E2 13856.075} C_VEL
LIN {X 0,Y 331.03,Z 728.021,A -85,B 0,C 180,E1 13851.663,E2 13851.663} C_VEL
LIN {X 0,Y 326.64,Z 718.81,A -85,B 0,C 180,E1 13847.54,E2 13847.54} C_VEL
LIN {X 0,Y 322.904,Z 710.813,A -85,B 0,C 180,E1 13843.633,E2 13843.633} C_VEL
LIN {X 0,Y 319.695,Z 704.73,A -85,B 0,C 180,E1 13840.258,E2 13840.258} C_VEL
LIN {X 0,Y 317.798,Z 700.823,A -85,B 0,C 180,E1 13838.012,E2 13838.012} C_VEL
LIN {X 0,Y 315.694,Z 696.529,A -85,B 0,C 180,E1 13835.361,E2 13835.361} C_VEL
LIN {X 0,Y 313.53,Z 692.135,A -85,B 0,C 180,E1 13832.439,E2 13832.439} C_VEL
LIN {X 0,Y 311.926,Z 689.132,A -85,B 0,C 180,E1 13830.207,E2 13830.207} C_VEL
LIN {X 0,Y 314.678,Z 689.969,A -85,B 0,C 180,E1 13829.337,E2 13829.337} C_VEL
LIN {X 0,Y 319.726,Z 699.946,A -85,B 0,C 180,E1 13826.605,E2 13826.605} C_VEL
LIN {X 0,Y 325.629,Z 713.29,A -85,B 0,C 180,E1 13823.437,E2 13823.437} C_VEL
LIN {X 0,Y 331.188,Z 727.772,A -85,B 0,C 180,E1 13820.429,E2 13820.429} C_VEL
LIN {X 0,Y 336.353,Z 743.637,A -85,B 0,C 180,E1 13817.56,E2 13817.56} C_VEL
LIN {X 0,Y 339.394,Z 755.276,A -85,B 0,C 180,E1 13815.659,E2 13815.659} C_VEL
LIN {X 0,Y 333.091,Z 803.63,A -85,B 0,C 180,E1 13811.213,E2 13811.213} C_VEL
LIN {X 0,Y 327.138,Z 853.33,A -85,B 0,C 180,E1 13806.69,E2 13806.69} C_VEL
LIN {X 0,Y 324.92,Z 875.175,A -85,B 0,C 180,E1 13804.779,E2 13804.779} C_VEL
LIN {X 0,Y 325.203,Z 881.742,A -85,B 0,C 180,E1 13804.567,E2 13804.567} C_VEL
LIN {X 0,Y 318.807,Z 1033.164,A -85,B 0,C 180,E1 13801.332,E2 13801.332} C_VEL
LIN {X 0,Y 318.14,Z 1053.417,A -85,B 0,C 180,E1 13800.722,E2 13800.722} C_VEL
LIN {X 0,Y 316.891,Z 1070.341,A -85,B 0,C 180,E1 13799.9,E2 13799.9} C_VEL
LIN {X 0,Y 314.934,Z 1087.052,A -85,B 0,C 180,E1 13798.747,E2 13798.747} C_VEL
LIN {X 0,Y 312.352,Z 1103.512,A -85,B 0,C 180,E1 13797.24,E2 13797.24} C_VEL
LIN {X 0,Y 309.564,Z 1117.999,A -85,B 0,C 180,E1 13795.541,E2 13795.541} C_VEL
LIN {X 0,Y 306.502,Z 1131.466,A -85,B 0,C 180,E1 13793.552,E2 13793.552} C_VEL
LIN {X 0,Y 303.323,Z 1143.902,A -85,B 0,C 180,E1 13791.258,E2 13791.258} C_VEL
LIN {X 0,Y 300.169,Z 1155.232,A -85,B 0,C 180,E1 13788.647,E2 13788.647} C_VEL
LIN {X 0,Y 297.3,Z 1164.972,A -85,B 0,C 180,E1 13785.805,E2 13785.805} C_VEL
LIN {X 0,Y 294.824,Z 1173.106,A -85,B 0,C 180,E1 13782.732,E2 13782.732} C_VEL
LIN {X 0,Y 292.86,Z 1179.674,A -85,B 0,C 180,E1 13779.429,E2 13779.429} C_VEL
LIN {X 0,Y 291.535,Z 1184.332,A -85,B 0,C 180,E1 13776.101,E2 13776.101} C_VEL
LIN {X 0,Y 290.742,Z 1187.304,A -85,B 0,C 180,E1 13772.56,E2 13772.56} C_VEL
LIN {X 0,Y 290.504,Z 1188.474,A -85,B 0,C 180,E1 13769.011,E2 13769.011} C_VEL
LIN {X 0,Y 290.783,Z 1187.866,A -85,B 0,C 180,E1 13765.461,E2 13765.461} C_VEL
LIN {X 0,Y 291.618,Z 1185.364,A -85,B 0,C 180,E1 13761.916,E2 13761.916} C_VEL
LIN {X 0,Y 293.106,Z 1180.964,A -85,B 0,C 180,E1 13758.386,E2 13758.386} C_VEL
LIN {X 0,Y 295.183,Z 1174.897,A -85,B 0,C 180,E1 13755.079,E2 13755.079} C_VEL
LIN {X 0,Y 297.766,Z 1167.19,A -85,B 0,C 180,E1 13752.003,E2 13752.003} C_VEL
LIN {X 0,Y 300.936,Z 1157.457,A -85,B 0,C 180,E1 13749.012,E2 13749.012} C_VEL
LIN {X 0,Y 304.302,Z 1146.458,A -85,B 0,C 180,E1 13746.365,E2 13746.365} C_VEL
LIN {X 0,Y 307.764,Z 1133.924,A -85,B 0,C 180,E1 13743.983,E2 13743.983} C_VEL
LIN {X 0,Y 311.126,Z 1120.269,A -85,B 0,C 180,E1 13741.91,E2 13741.91} C_VEL
LIN {X 0,Y 314.067,Z 1106.344,A -85,B 0,C 180,E1 13740.219,E2 13740.219} C_VEL
LIN {X 0,Y 316.628,Z 1091.625,A -85,B 0,C 180,E1 13738.806,E2 13738.806} C_VEL
LIN {X 0,Y 318.779,Z 1075.448,A -85,B 0,C 180,E1 13737.614,E2 13737.614} C_VEL
LIN {X 0,Y 320.372,Z 1057.867,A -85,B 0,C 180,E1 13736.672,E2 13736.672} C_VEL
LIN {X 0,Y 321.2,Z 1040.237,A -85,B 0,C 180,E1 13736.056,E2 13736.056} C_VEL
LIN {X 0,Y 323.168,Z 986.036,A -85,B 0,C 180,E1 13734.854,E2 13734.854} C_VEL
LIN {X 0,Y 325.503,Z 937.081,A -85,B 0,C 180,E1 13733.801,E2 13733.801} C_VEL
LIN {X 0,Y 327.162,Z 937.592,A -85,B 0,C 180,E1 13733.525,E2 13733.525} C_VEL
LIN {X 0,Y 329.415,Z 935.907,A -85,B 0,C 180,E1 13733.298,E2 13733.298} C_VEL
LIN {X 0,Y 332.626,Z 930.874,A -85,B 0,C 180,E1 13733.13,E2 13733.13} C_VEL
LIN {X 0,Y 336.623,Z 921.108,A -85,B 0,C 180,E1 13733.12,E2 13733.12} C_VEL
LIN {X 0,Y 337.272,Z 919.745,A -85,B 0,C 180,E1 13733.104,E2 13733.104} C_VEL
LIN {X 0,Y 340.903,Z 916.307,A -85,B 0,C 180,E1 13732.773,E2 13732.773} C_VEL
LIN {X 0,Y 344.839,Z 910.039,A -85,B 0,C 180,E1 13732.558,E2 13732.558} C_VEL
LIN {X 0,Y 349.069,Z 899.867,A -85,B 0,C 180,E1 13732.51,E2 13732.51} C_VEL
LIN {X 0,Y 354.166,Z 893.433,A -85,B 0,C 180,E1 13732.128,E2 13732.128} C_VEL
LIN {X 0,Y 357.373,Z 888.027,A -85,B 0,C 180,E1 13731.956,E2 13731.956} C_VEL
LIN {X 0,Y 363.418,Z 882.883,A -85,B 0,C 180,E1 13731.374,E2 13731.374} C_VEL
LIN {X 0,Y 364.505,Z 882.141,A -85,B 0,C 180,E1 13731.262,E2 13731.262} C_VEL
LIN {X 0,Y 351.459,Z 976.022,A -85,B 0,C 180,E1 13728.222,E2 13728.222} C_VEL
LIN {X 0,Y 349.68,Z 983.516,A -85,B 0,C 180,E1 13728.052,E2 13728.052} C_VEL
LIN {X 0,Y 341.98,Z 1003.28,A -85,B 0,C 180,E1 13727.876,E2 13727.876} C_VEL
LIN {X 0,Y 340.428,Z 1009.614,A -85,B 0,C 180,E1 13727.655,E2 13727.655} C_VEL
LIN {X 0,Y 336.537,Z 1032.319,A -85,B 0,C 180,E1 13726.465,E2 13726.465} C_VEL
LIN {X 0,Y 331.824,Z 1055.025,A -85,B 0,C 180,E1 13724.961,E2 13724.961} C_VEL
LIN {X 0,Y 326.578,Z 1076.768,A -85,B 0,C 180,E1 13723.18,E2 13723.18} C_VEL
LIN {X 0,Y 320.947,Z 1097.696,A -85,B 0,C 180,E1 13721.099,E2 13721.099} C_VEL
LIN {X 0,Y 314.853,Z 1118.326,A -85,B 0,C 180,E1 13718.624,E2 13718.624} C_VEL
LIN {X 0,Y 309.155,Z 1136.357,A -85,B 0,C 180,E1 13716.041,E2 13716.041} C_VEL
LIN {X 0,Y 303.241,Z 1154.325,A -85,B 0,C 180,E1 13712.961,E2 13712.961} C_VEL
LIN {X 0,Y 297.707,Z 1170.708,A -85,B 0,C 180,E1 13709.586,E2 13709.586} C_VEL
LIN {X 0,Y 293.004,Z 1184.844,A -85,B 0,C 180,E1 13706.118,E2 13706.118} C_VEL
LIN {X 0,Y 288.734,Z 1198.321,A -85,B 0,C 180,E1 13702.177,E2 13702.177} C_VEL
LIN {X 0,Y 285.449,Z 1209.762,A -85,B 0,C 180,E1 13698.165,E2 13698.165} C_VEL
LIN {X 0,Y 282.99,Z 1219.705,A -85,B 0,C 180,E1 13693.902,E2 13693.902} C_VEL
LIN {X 0,Y 281.458,Z 1227.816,A -85,B 0,C 180,E1 13689.612,E2 13689.612} C_VEL
LIN {X 0,Y 280.657,Z 1234.316,A -85,B 0,C 180,E1 13685.315,E2 13685.315} C_VEL
LIN {X 0,Y 280.401,Z 1239.005,A -85,B 0,C 180,E1 13681.226,E2 13681.226} C_VEL
LIN {X 0,Y 280.425,Z 1242.563,A -85,B 0,C 180,E1 13676.934,E2 13676.934} C_VEL
LIN {X 0,Y 280.723,Z 1244.705,A -85,B 0,C 180,E1 13672.839,E2 13672.839} C_VEL
LIN {X 0,Y 281.614,Z 1245.735,A -85,B 0,C 180,E1 13668.116,E2 13668.116} C_VEL
LIN {X 0,Y 283.572,Z 1245.279,A -85,B 0,C 180,E1 13663.194,E2 13663.194} C_VEL
LIN {X 0,Y 287.134,Z 1243.175,A -85,B 0,C 180,E1 13658.123,E2 13658.123} C_VEL
LIN {X 0,Y 292.769,Z 1239.224,A -85,B 0,C 180,E1 13652.984,E2 13652.984} C_VEL
LIN {X 0,Y 300.836,Z 1233.221,A -85,B 0,C 180,E1 13647.873,E2 13647.873} C_VEL
LIN {X 0,Y 310.854,Z 1225.59,A -85,B 0,C 180,E1 13643.222,E2 13643.222} C_VEL
LIN {X 0,Y 322.883,Z 1216.27,A -85,B 0,C 180,E1 13638.965,E2 13638.965} C_VEL
LIN {X 0,Y 337.629,Z 1204.712,A -85,B 0,C 180,E1 13634.944,E2 13634.944} C_VEL
LIN {X 0,Y 339.993,Z 1202.917,A -85,B 0,C 180,E1 13634.371,E2 13634.371} C_VEL
LIN {X 0,Y 323.338,Z 1216.458,A -85,B 0,C 180,E1 13630.733,E2 13630.733} C_VEL
LIN {X 0,Y 308.052,Z 1231.237,A -85,B 0,C 180,E1 13625.982,E2 13625.982} C_VEL
LIN {X 0,Y 296.666,Z 1244.473,A -85,B 0,C 180,E1 13620.82,E2 13620.82} C_VEL
LIN {X 0,Y 288.963,Z 1255.224,A -85,B 0,C 180,E1 13615.631,E2 13615.631} C_VEL
LIN {X 0,Y 284.169,Z 1263.37,A -85,B 0,C 180,E1 13610.604,E2 13610.604} C_VEL
LIN {X 0,Y 281.556,Z 1269.062,A -85,B 0,C 180,E1 13605.872,E2 13605.872} C_VEL
LIN {X 0,Y 280.423,Z 1272.744,A -85,B 0,C 180,E1 13601.312,E2 13601.312} C_VEL
LIN {X 0,Y 280.258,Z 1274.541,A -85,B 0,C 180,E1 13596.97,E2 13596.97} C_VEL
LIN {X 0,Y 280.483,Z 1274.645,A -85,B 0,C 180,E1 13593.068,E2 13593.068} C_VEL
LIN {X 0,Y 280.692,Z 1273.338,A -85,B 0,C 180,E1 13589.39,E2 13589.39} C_VEL
LIN {X 0,Y 280.698,Z 1270.571,A -85,B 0,C 180,E1 13585.713,E2 13585.713} C_VEL
LIN {X 0,Y 280.649,Z 1266.296,A -85,B 0,C 180,E1 13582.016,E2 13582.016} C_VEL
LIN {X 0,Y 280.831,Z 1260.122,A -85,B 0,C 180,E1 13578.085,E2 13578.085} C_VEL
LIN {X 0,Y 281.576,Z 1251.733,A -85,B 0,C 180,E1 13573.923,E2 13573.923} C_VEL
LIN {X 0,Y 283.1,Z 1241.403,A -85,B 0,C 180,E1 13569.753,E2 13569.753} C_VEL
LIN {X 0,Y 285.591,Z 1228.948,A -85,B 0,C 180,E1 13565.602,E2 13565.602} C_VEL
LIN {X 0,Y 289.249,Z 1213.95,A -85,B 0,C 180,E1 13561.407,E2 13561.407} C_VEL
LIN {X 0,Y 294.144,Z 1196.339,A -85,B 0,C 180,E1 13557.287,E2 13557.287} C_VEL
LIN {X 0,Y 299.826,Z 1177.594,A -85,B 0,C 180,E1 13553.59,E2 13553.59} C_VEL
LIN {X 0,Y 306.427,Z 1156.818,A -85,B 0,C 180,E1 13550.123,E2 13550.123} C_VEL
LIN {X 0,Y 314.109,Z 1133.15,A -85,B 0,C 180,E1 13546.816,E2 13546.816} C_VEL
LIN {X 0,Y 323.187,Z 1105.343,A -85,B 0,C 180,E1 13543.622,E2 13543.622} C_VEL
LIN {X 0,Y 331.474,Z 1079.886,A -85,B 0,C 180,E1 13541.179,E2 13541.179} C_VEL
LIN {X 0,Y 339.976,Z 1053.036,A -85,B 0,C 180,E1 13539.069,E2 13539.069} C_VEL
LIN {X 0,Y 348.222,Z 1025.739,A -85,B 0,C 180,E1 13537.313,E2 13537.313} C_VEL
LIN {X 0,Y 355.91,Z 998.016,A -85,B 0,C 180,E1 13535.859,E2 13535.859} C_VEL
LIN {X 0,Y 356.723,Z 994.101,A -85,B 0,C 180,E1 13535.664,E2 13535.664} C_VEL
LIN {X 0,Y 352.315,Z 972.897,A -85,B 0,C 180,E1 13533.505,E2 13533.505} C_VEL
LIN {X 0,Y 348.684,Z 949.31,A -85,B 0,C 180,E1 13531.364,E2 13531.364} C_VEL
LIN {X 0,Y 345.998,Z 924.473,A -85,B 0,C 180,E1 13529.389,E2 13529.389} C_VEL
LIN {X 0,Y 344.416,Z 897.488,A -85,B 0,C 180,E1 13527.502,E2 13527.502} C_VEL
LIN {X 0,Y 344.279,Z 885.772,A -85,B 0,C 180,E1 13526.754,E2 13526.754} C_VEL
LIN {X 0,Y 353.983,Z 851.27,A -85,B 0,C 180,E1 13522.539,E2 13522.539} C_VEL
LIN {X 0,Y 361.743,Z 824.426,A -85,B 0,C 180,E1 13519.246,E2 13519.246} C_VEL
LIN {X 0,Y 355.966,Z 807.818,A -85,B 0,C 180,E1 13515.31,E2 13515.31} C_VEL
LIN {X 0,Y 350.504,Z 793.213,A -85,B 0,C 180,E1 13511.519,E2 13511.519} C_VEL
LIN {X 0,Y 345.21,Z 779.518,A -85,B 0,C 180,E1 13507.657,E2 13507.657} C_VEL
LIN {X 0,Y 339.985,Z 766.76,A -85,B 0,C 180,E1 13503.71,E2 13503.71} C_VEL
LIN {X 0,Y 334.923,Z 754.825,A -85,B 0,C 180,E1 13499.658,E2 13499.658} C_VEL
LIN {X 0,Y 330.176,Z 744.061,A -85,B 0,C 180,E1 13495.658,E2 13495.658} C_VEL
LIN {X 0,Y 325.402,Z 733.436,A -85,B 0,C 180,E1 13491.34,E2 13491.34} C_VEL
LIN {X 0,Y 321.336,Z 724.766,A -85,B 0,C 180,E1 13487.419,E2 13487.419} C_VEL
LIN {X 0,Y 317.393,Z 716.409,A -85,B 0,C 180,E1 13483.264,E2 13483.264} C_VEL
LIN {X 0,Y 314.236,Z 710.257,A -85,B 0,C 180,E1 13479.822,E2 13479.822} C_VEL
LIN {X 0,Y 312.571,Z 706.795,A -85,B 0,C 180,E1 13477.823,E2 13477.823} C_VEL
LIN {X 0,Y 310.549,Z 702.607,A -85,B 0,C 180,E1 13475.218,E2 13475.218} C_VEL
LIN {X 0,Y 308.291,Z 698.078,A -85,B 0,C 180,E1 13472.158,E2 13472.158} C_VEL
LIN {X 0,Y 307.173,Z 696.039,A -85,B 0,C 180,E1 13470.559,E2 13470.559} C_VEL
LIN {X 0,Y 310.453,Z 696.875,A -85,B 0,C 180,E1 13469.518,E2 13469.518} C_VEL
LIN {X 0,Y 316.082,Z 708.657,A -85,B 0,C 180,E1 13466.296,E2 13466.296} C_VEL
LIN {X 0,Y 322.091,Z 722.981,A -85,B 0,C 180,E1 13462.969,E2 13462.969} C_VEL
LIN {X 0,Y 327.526,Z 738.228,A -85,B 0,C 180,E1 13459.897,E2 13459.897} C_VEL
LIN {X 0,Y 332.101,Z 753.844,A -85,B 0,C 180,E1 13457.121,E2 13457.121} C_VEL
LIN {X 0,Y 333.116,Z 758.893,A -85,B 0,C 180,E1 13456.331,E2 13456.331} C_VEL
LIN {X 0,Y 326.616,Z 807.206,A -85,B 0,C 180,E1 13451.861,E2 13451.861} C_VEL
LIN {X 0,Y 320.524,Z 856.336,A -85,B 0,C 180,E1 13447.351,E2 13447.351} C_VEL
LIN {X 0,Y 318.449,Z 876.142,A -85,B 0,C 180,E1 13445.606,E2 13445.606} C_VEL
LIN {X 0,Y 318.706,Z 882.735,A -85,B 0,C 180,E1 13445.389,E2 13445.389} C_VEL
LIN {X 0,Y 312.085,Z 1033.535,A -85,B 0,C 180,E1 13442.117,E2 13442.117} C_VEL
LIN {X 0,Y 311.396,Z 1053.8,A -85,B 0,C 180,E1 13441.503,E2 13441.503} C_VEL
LIN {X 0,Y 310.115,Z 1070.709,A -85,B 0,C 180,E1 13440.676,E2 13440.676} C_VEL
LIN {X 0,Y 308.165,Z 1087.075,A -85,B 0,C 180,E1 13439.547,E2 13439.547} C_VEL
LIN {X 0,Y 305.634,Z 1102.854,A -85,B 0,C 180,E1 13438.102,E2 13438.102} C_VEL
LIN {X 0,Y 302.722,Z 1117.635,A -85,B 0,C 180,E1 13436.372,E2 13436.372} C_VEL
LIN {X 0,Y 299.529,Z 1131.414,A -85,B 0,C 180,E1 13434.344,E2 13434.344} C_VEL
LIN {X 0,Y 296.195,Z 1144.026,A -85,B 0,C 180,E1 13432.003,E2 13432.003} C_VEL
LIN {X 0,Y 292.877,Z 1155.497,A -85,B 0,C 180,E1 13429.336,E2 13429.336} C_VEL
LIN {X 0,Y 289.851,Z 1165.396,A -85,B 0,C 180,E1 13426.429,E2 13426.429} C_VEL
LIN {X 0,Y 287.227,Z 1173.651,A -85,B 0,C 180,E1 13423.28,E2 13423.28} C_VEL
LIN {X 0,Y 285.128,Z 1180.314,A -85,B 0,C 180,E1 13419.892,E2 13419.892} C_VEL
LIN {X 0,Y 283.702,Z 1185.071,A -85,B 0,C 180,E1 13416.473,E2 13416.473} C_VEL
LIN {X 0,Y 282.87,Z 1188.047,A -85,B 0,C 180,E1 13413.037,E2 13413.037} C_VEL
LIN {X 0,Y 282.562,Z 1189.383,A -85,B 0,C 180,E1 13409.389,E2 13409.389} C_VEL
LIN {X 0,Y 282.795,Z 1188.948,A -85,B 0,C 180,E1 13405.739,E2 13405.739} C_VEL
LIN {X 0,Y 283.614,Z 1186.696,A -85,B 0,C 180,E1 13402.094,E2 13402.094} C_VEL
LIN {X 0,Y 285,Z 1182.765,A -85,B 0,C 180,E1 13398.667,E2 13398.667} C_VEL
LIN {X 0,Y 287.054,Z 1177.008,A -85,B 0,C 180,E1 13395.267,E2 13395.267} C_VEL
LIN {X 0,Y 289.648,Z 1169.729,A -85,B 0,C 180,E1 13392.105,E2 13392.105} C_VEL
LIN {X 0,Y 292.665,Z 1160.919,A -85,B 0,C 180,E1 13389.185,E2 13389.185} C_VEL
LIN {X 0,Y 295.986,Z 1150.654,A -85,B 0,C 180,E1 13386.505,E2 13386.505} C_VEL
LIN {X 0,Y 299.481,Z 1138.933,A -85,B 0,C 180,E1 13384.061,E2 13384.061} C_VEL
LIN {X 0,Y 303.04,Z 1125.632,A -85,B 0,C 180,E1 13381.844,E2 13381.844} C_VEL
LIN {X 0,Y 306.364,Z 1111.083,A -85,B 0,C 180,E1 13379.933,E2 13379.933} C_VEL
LIN {X 0,Y 309.338,Z 1095.391,A -85,B 0,C 180,E1 13378.312,E2 13378.312} C_VEL
LIN {X 0,Y 311.703,Z 1079.365,A -85,B 0,C 180,E1 13377.039,E2 13377.039} C_VEL
LIN {X 0,Y 313.446,Z 1062.274,A -85,B 0,C 180,E1 13376.049,E2 13376.049} C_VEL
LIN {X 0,Y 314.473,Z 1044.113,A -85,B 0,C 180,E1 13375.347,E2 13375.347} C_VEL
LIN {X 0,Y 316.268,Z 994.597,A -85,B 0,C 180,E1 13374.199,E2 13374.199} C_VEL
LIN {X 0,Y 317.895,Z 960.399,A -85,B 0,C 180,E1 13373.467,E2 13373.467} C_VEL
LIN {X 0,Y 319.134,Z 961.183,A -85,B 0,C 180,E1 13373.24,E2 13373.24} C_VEL
LIN {X 0,Y 321.139,Z 960.341,A -85,B 0,C 180,E1 13373.006,E2 13373.006} C_VEL
LIN {X 0,Y 324.152,Z 956.456,A -85,B 0,C 180,E1 13372.811,E2 13372.811} C_VEL
LIN {X 0,Y 328.036,Z 948.281,A -85,B 0,C 180,E1 13372.758,E2 13372.758} C_VEL
LIN {X 0,Y 329.679,Z 944.066,A -85,B 0,C 180,E1 13372.775,E2 13372.775} C_VEL
LIN {X 0,Y 333.409,Z 940.762,A -85,B 0,C 180,E1 13372.441,E2 13372.441} C_VEL
LIN {X 0,Y 337.248,Z 934.909,A -85,B 0,C 180,E1 13372.235,E2 13372.235} C_VEL
LIN {X 0,Y 341.532,Z 925.014,A -85,B 0,C 180,E1 13372.196,E2 13372.196} C_VEL
LIN {X 0,Y 347.105,Z 918.06,A -85,B 0,C 180,E1 13371.801,E2 13371.801} C_VEL
LIN {X 0,Y 351.534,Z 909.707,A -85,B 0,C 180,E1 13371.632,E2 13371.632} C_VEL
LIN {X 0,Y 354.302,Z 903.256,A -85,B 0,C 180,E1 13371.592,E2 13371.592} C_VEL
LIN {X 0,Y 355.6,Z 901.926,A -85,B 0,C 180,E1 13371.481,E2 13371.481} C_VEL
LIN {X 0,Y 343.674,Z 986.058,A -85,B 0,C 180,E1 13368.619,E2 13368.619} C_VEL
LIN {X 0,Y 340.428,Z 1009.614,A -85,B 0,C 180,E1 13367.655,E2 13367.655} C_VEL
LIN {X 0,Y 338.335,Z 1016.943,A -85,B 0,C 180,E1 13367.412,E2 13367.412} C_VEL
LIN {X 0,Y 329.995,Z 1035.091,A -85,B 0,C 180,E1 13366.965,E2 13366.965} C_VEL
LIN {X 0,Y 327.815,Z 1042.24,A -85,B 0,C 180,E1 13366.59,E2 13366.59} C_VEL
LIN {X 0,Y 322.999,Z 1063.469,A -85,B 0,C 180,E1 13365.034,E2 13365.034} C_VEL
LIN {X 0,Y 317.319,Z 1085.556,A -85,B 0,C 180,E1 13363.052,E2 13363.052} C_VEL
LIN {X 0,Y 311.383,Z 1106.227,A -85,B 0,C 180,E1 13360.804,E2 13360.804} C_VEL
LIN {X 0,Y 305.291,Z 1125.797,A -85,B 0,C 180,E1 13358.244,E2 13358.244} C_VEL
LIN {X 0,Y 298.959,Z 1144.945,A -85,B 0,C 180,E1 13355.216,E2 13355.216} C_VEL
LIN {X 0,Y 293.355,Z 1161.277,A -85,B 0,C 180,E1 13352.122,E2 13352.122} C_VEL
LIN {X 0,Y 287.814,Z 1177.399,A -85,B 0,C 180,E1 13348.481,E2 13348.481} C_VEL
LIN {X 0,Y 283.075,Z 1191.593,A -85,B 0,C 180,E1 13344.633,E2 13344.633} C_VEL
LIN {X 0,Y 279.166,Z 1204.159,A -85,B 0,C 180,E1 13340.549,E2 13340.549} C_VEL
LIN {X 0,Y 276.128,Z 1215.172,A -85,B 0,C 180,E1 13336.19,E2 13336.19} C_VEL
LIN {X 0,Y 274.112,Z 1224.25,A -85,B 0,C 180,E1 13331.787,E2 13331.787} C_VEL
LIN {X 0,Y 272.914,Z 1231.911,A -85,B 0,C 180,E1 13327.156,E2 13327.156} C_VEL
LIN {X 0,Y 272.451,Z 1237.625,A -85,B 0,C 180,E1 13322.735,E2 13322.735} C_VEL
LIN {X 0,Y 272.392,Z 1241.584,A -85,B 0,C 180,E1 13318.528,E2 13318.528} C_VEL
LIN {X 0,Y 272.61,Z 1244.53,A -85,B 0,C 180,E1 13314.105,E2 13314.105} C_VEL
LIN {X 0,Y 273.247,Z 1246.079,A -85,B 0,C 180,E1 13309.671,E2 13309.671} C_VEL
LIN {X 0,Y 274.986,Z 1246.404,A -85,B 0,C 180,E1 13304.391,E2 13304.391} C_VEL
LIN {X 0,Y 278.294,Z 1245.049,A -85,B 0,C 180,E1 13299.099,E2 13299.099} C_VEL
LIN {X 0,Y 283.592,Z 1241.983,A -85,B 0,C 180,E1 13293.85,E2 13293.85} C_VEL
LIN {X 0,Y 291.091,Z 1237.17,A -85,B 0,C 180,E1 13288.756,E2 13288.756} C_VEL
LIN {X 0,Y 301.219,Z 1230.36,A -85,B 0,C 180,E1 13283.781,E2 13283.781} C_VEL
LIN {X 0,Y 313.693,Z 1221.728,A -85,B 0,C 180,E1 13279.199,E2 13279.199} C_VEL
LIN {X 0,Y 329.032,Z 1210.946,A -85,B 0,C 180,E1 13274.922,E2 13274.922} C_VEL
LIN {X 0,Y 330.856,Z 1209.702,A -85,B 0,C 180,E1 13274.466,E2 13274.466} C_VEL
LIN {X 0,Y 314.288,Z 1222.376,A -85,B 0,C 180,E1 13270.71,E2 13270.71} C_VEL
LIN {X 0,Y 298.649,Z 1236.538,A -85,B 0,C 180,E1 13265.633,E2 13265.633} C_VEL
LIN {X 0,Y 287.161,Z 1249.016,A -85,B 0,C 180,E1 13260.096,E2 13260.096} C_VEL
LIN {X 0,Y 280.015,Z 1258.328,A -85,B 0,C 180,E1 13254.906,E2 13254.906} C_VEL
LIN {X 0,Y 275.511,Z 1265.457,A -85,B 0,C 180,E1 13249.728,E2 13249.728} C_VEL
LIN {X 0,Y 273.179,Z 1270.258,A -85,B 0,C 180,E1 13244.848,E2 13244.848} C_VEL
LIN {X 0,Y 272.317,Z 1273.067,A -85,B 0,C 180,E1 13240.249,E2 13240.249} C_VEL
LIN {X 0,Y 272.323,Z 1274.109,A -85,B 0,C 180,E1 13235.904,E2 13235.904} C_VEL
LIN {X 0,Y 272.588,Z 1273.65,A -85,B 0,C 180,E1 13232.105,E2 13232.105} C_VEL
LIN {X 0,Y 272.762,Z 1271.889,A -85,B 0,C 180,E1 13228.532,E2 13228.532} C_VEL
LIN {X 0,Y 272.745,Z 1268.823,A -85,B 0,C 180,E1 13224.955,E2 13224.955} C_VEL
LIN {X 0,Y 272.711,Z 1263.817,A -85,B 0,C 180,E1 13220.932,E2 13220.932} C_VEL
LIN {X 0,Y 273.01,Z 1257.093,A -85,B 0,C 180,E1 13216.878,E2 13216.878} C_VEL
LIN {X 0,Y 273.906,Z 1248.626,A -85,B 0,C 180,E1 13212.804,E2 13212.804} C_VEL
LIN {X 0,Y 275.719,Z 1237.682,A -85,B 0,C 180,E1 13208.517,E2 13208.517} C_VEL
LIN {X 0,Y 278.546,Z 1224.679,A -85,B 0,C 180,E1 13204.259,E2 13204.259} C_VEL
LIN {X 0,Y 282.517,Z 1209.363,A -85,B 0,C 180,E1 13200.068,E2 13200.068} C_VEL
LIN {X 0,Y 287.559,Z 1192.107,A -85,B 0,C 180,E1 13196.08,E2 13196.08} C_VEL
LIN {X 0,Y 293.782,Z 1172.289,A -85,B 0,C 180,E1 13192.224,E2 13192.224} C_VEL
LIN {X 0,Y 301.236,Z 1149.584,A -85,B 0,C 180,E1 13188.537,E2 13188.537} C_VEL
LIN {X 0,Y 309.453,Z 1125,A -85,B 0,C 180,E1 13185.224,E2 13185.224} C_VEL
LIN {X 0,Y 317.988,Z 1099.375,A -85,B 0,C 180,E1 13182.363,E2 13182.363} C_VEL
LIN {X 0,Y 326.936,Z 1072.411,A -85,B 0,C 180,E1 13179.862,E2 13179.862} C_VEL
LIN {X 0,Y 335.458,Z 1045.976,A -85,B 0,C 180,E1 13177.831,E2 13177.831} C_VEL
LIN {X 0,Y 343.666,Z 1019.086,A -85,B 0,C 180,E1 13176.164,E2 13176.164} C_VEL
LIN {X 0,Y 349.935,Z 995.915,A -85,B 0,C 180,E1 13174.943,E2 13174.943} C_VEL
LIN {X 0,Y 345.354,Z 972.029,A -85,B 0,C 180,E1 13172.485,E2 13172.485} C_VEL
LIN {X 0,Y 342.284,Z 949.724,A -85,B 0,C 180,E1 13170.429,E2 13170.429} C_VEL
LIN {X 0,Y 339.82,Z 922.968,A -85,B 0,C 180,E1 13168.277,E2 13168.277} C_VEL
LIN {X 0,Y 338.628,Z 895.129,A -85,B 0,C 180,E1 13166.337,E2 13166.337} C_VEL
LIN {X 0,Y 338.695,Z 883.493,A -85,B 0,C 180,E1 13165.579,E2 13165.579} C_VEL
LIN {X 0,Y 348.663,Z 849.338,A -85,B 0,C 180,E1 13161.359,E2 13161.359} C_VEL
LIN {X 0,Y 355.02,Z 827.922,A -85,B 0,C 180,E1 13158.728,E2 13158.728} C_VEL
LIN {X 0,Y 349.807,Z 812.724,A -85,B 0,C 180,E1 13155.077,E2 13155.077} C_VEL
LIN {X 0,Y 344.609,Z 798.625,A -85,B 0,C 180,E1 13151.379,E2 13151.379} C_VEL
LIN {X 0,Y 339.122,Z 784.266,A -85,B 0,C 180,E1 13147.284,E2 13147.284} C_VEL
LIN {X 0,Y 333.727,Z 770.962,A -85,B 0,C 180,E1 13143.091,E2 13143.091} C_VEL
LIN {X 0,Y 328.436,Z 758.435,A -85,B 0,C 180,E1 13138.779,E2 13138.779} C_VEL
LIN {X 0,Y 323.548,Z 747.211,A -85,B 0,C 180,E1 13134.502,E2 13134.502} C_VEL
LIN {X 0,Y 318.965,Z 737.216,A -85,B 0,C 180,E1 13130.254,E2 13130.254} C_VEL
LIN {X 0,Y 315.141,Z 729.011,A -85,B 0,C 180,E1 13126.421,E2 13126.421} C_VEL
LIN {X 0,Y 311.655,Z 721.586,A -85,B 0,C 180,E1 13122.64,E2 13122.64} C_VEL
LIN {X 0,Y 309.08,Z 716.386,A -85,B 0,C 180,E1 13119.736,E2 13119.736} C_VEL
LIN {X 0,Y 307.258,Z 712.626,A -85,B 0,C 180,E1 13117.54,E2 13117.54} C_VEL
LIN {X 0,Y 305.129,Z 708.281,A -85,B 0,C 180,E1 13114.786,E2 13114.786} C_VEL
LIN {X 0,Y 303.252,Z 704.279,A -85,B 0,C 180,E1 13112.079,E2 13112.079} C_VEL
LIN {X 0,Y 302.505,Z 702.949,A -85,B 0,C 180,E1 13110.929,E2 13110.929} C_VEL
LIN {X 0,Y 306.377,Z 704.033,A -85,B 0,C 180,E1 13109.611,E2 13109.611} C_VEL
LIN {X 0,Y 311.813,Z 716.183,A -85,B 0,C 180,E1 13106.306,E2 13106.306} C_VEL
LIN {X 0,Y 317.277,Z 729.625,A -85,B 0,C 180,E1 13103.17,E2 13103.17} C_VEL
LIN {X 0,Y 322.391,Z 744.47,A -85,B 0,C 180,E1 13100.174,E2 13100.174} C_VEL
LIN {X 0,Y 326.965,Z 760.956,A -85,B 0,C 180,E1 13097.242,E2 13097.242} C_VEL
LIN {X 0,Y 326.866,Z 763.306,A -85,B 0,C 180,E1 13096.975,E2 13096.975} C_VEL
LIN {X 0,Y 320.039,Z 811.833,A -85,B 0,C 180,E1 13092.438,E2 13092.438} C_VEL
LIN {X 0,Y 313.708,Z 861.524,A -85,B 0,C 180,E1 13087.844,E2 13087.844} C_VEL
LIN {X 0,Y 312.045,Z 877.092,A -85,B 0,C 180,E1 13086.468,E2 13086.468} C_VEL
LIN {X 0,Y 312.283,Z 883.6,A -85,B 0,C 180,E1 13086.249,E2 13086.249} C_VEL
LIN {X 0,Y 305.423,Z 1033.904,A -85,B 0,C 180,E1 13082.936,E2 13082.936} C_VEL
LIN {X 0,Y 304.712,Z 1054.183,A -85,B 0,C 180,E1 13082.318,E2 13082.318} C_VEL
LIN {X 0,Y 303.35,Z 1071.585,A -85,B 0,C 180,E1 13081.458,E2 13081.458} C_VEL
LIN {X 0,Y 301.292,Z 1088.181,A -85,B 0,C 180,E1 13080.291,E2 13080.291} C_VEL
LIN {X 0,Y 298.662,Z 1103.932,A -85,B 0,C 180,E1 13078.819,E2 13078.819} C_VEL
LIN {X 0,Y 295.638,Z 1118.692,A -85,B 0,C 180,E1 13077.055,E2 13077.055} C_VEL
LIN {X 0,Y 292.304,Z 1132.511,A -85,B 0,C 180,E1 13074.974,E2 13074.974} C_VEL
LIN {X 0,Y 288.853,Z 1145.045,A -85,B 0,C 180,E1 13072.593,E2 13072.593} C_VEL
LIN {X 0,Y 285.399,Z 1156.506,A -85,B 0,C 180,E1 13069.864,E2 13069.864} C_VEL
LIN {X 0,Y 282.244,Z 1166.395,A -85,B 0,C 180,E1 13066.885,E2 13066.885} C_VEL
LIN {X 0,Y 279.503,Z 1174.639,A -85,B 0,C 180,E1 13063.654,E2 13063.654} C_VEL
LIN {X 0,Y 277.272,Z 1181.408,A -85,B 0,C 180,E1 13060.104,E2 13060.104} C_VEL
LIN {X 0,Y 275.786,Z 1186.139,A -85,B 0,C 180,E1 13056.576,E2 13056.576} C_VEL
LIN {X 0,Y 274.906,Z 1189.117,A -85,B 0,C 180,E1 13052.916,E2 13052.916} C_VEL
LIN {X 0,Y 274.617,Z 1190.36,A -85,B 0,C 180,E1 13049.163,E2 13049.163} C_VEL
LIN {X 0,Y 274.902,Z 1189.833,A -85,B 0,C 180,E1 13045.408,E2 13045.408} C_VEL
LIN {X 0,Y 275.736,Z 1187.634,A -85,B 0,C 180,E1 13041.867,E2 13041.867} C_VEL
LIN {X 0,Y 277.199,Z 1183.696,A -85,B 0,C 180,E1 13038.343,E2 13038.343} C_VEL
LIN {X 0,Y 279.36,Z 1177.93,A -85,B 0,C 180,E1 13034.851,E2 13034.851} C_VEL
LIN {X 0,Y 282.081,Z 1170.641,A -85,B 0,C 180,E1 13031.608,E2 13031.608} C_VEL
LIN {X 0,Y 285.235,Z 1161.815,A -85,B 0,C 180,E1 13028.616,E2 13028.616} C_VEL
LIN {X 0,Y 288.702,Z 1151.537,A -85,B 0,C 180,E1 13025.875,E2 13025.875} C_VEL
LIN {X 0,Y 292.344,Z 1139.802,A -85,B 0,C 180,E1 13023.379,E2 13023.379} C_VEL
LIN {X 0,Y 296.046,Z 1126.475,A -85,B 0,C 180,E1 13021.117,E2 13021.117} C_VEL
LIN {X 0,Y 299.501,Z 1111.896,A -85,B 0,C 180,E1 13019.169,E2 13019.169} C_VEL
LIN {X 0,Y 302.591,Z 1096.169,A -85,B 0,C 180,E1 13017.52,E2 13017.52} C_VEL
LIN {X 0,Y 305.086,Z 1079.787,A -85,B 0,C 180,E1 13016.204,E2 13016.204} C_VEL
LIN {X 0,Y 306.888,Z 1062.511,A -85,B 0,C 180,E1 13015.201,E2 13015.201} C_VEL
LIN {X 0,Y 307.931,Z 1044.482,A -85,B 0,C 180,E1 13014.502,E2 13014.502} C_VEL
LIN {X 0,Y 309.83,Z 994.509,A -85,B 0,C 180,E1 13013.328,E2 13013.328} C_VEL
LIN {X 0,Y 310.416,Z 983.19,A -85,B 0,C 180,E1 13013.075,E2 13013.075} C_VEL
LIN {X 0,Y 311.474,Z 983.954,A -85,B 0,C 180,E1 13012.875,E2 13012.875} C_VEL
LIN {X 0,Y 313.452,Z 983.405,A -85,B 0,C 180,E1 13012.633,E2 13012.633} C_VEL
LIN {X 0,Y 316.366,Z 980.117,A -85,B 0,C 180,E1 13012.438,E2 13012.438} C_VEL
LIN {X 0,Y 320.105,Z 972.837,A -85,B 0,C 180,E1 13012.377,E2 13012.377} C_VEL
LIN {X 0,Y 322.122,Z 967.715,A -85,B 0,C 180,E1 13012.412,E2 13012.412} C_VEL
LIN {X 0,Y 325.835,Z 964.623,A -85,B 0,C 180,E1 13012.087,E2 13012.087} C_VEL
LIN {X 0,Y 329.784,Z 958.893,A -85,B 0,C 180,E1 13011.886,E2 13011.886} C_VEL
LIN {X 0,Y 333.966,Z 949.609,A -85,B 0,C 180,E1 13011.85,E2 13011.85} C_VEL
LIN {X 0,Y 334.896,Z 948.3,A -85,B 0,C 180,E1 13011.798,E2 13011.798} C_VEL
LIN {X 0,Y 339.469,Z 942.97,A -85,B 0,C 180,E1 13011.478,E2 13011.478} C_VEL
LIN {X 0,Y 343.928,Z 934.992,A -85,B 0,C 180,E1 13011.316,E2 13011.316} C_VEL
LIN {X 0,Y 344.796,Z 933.182,A -85,B 0,C 180,E1 13011.296,E2 13011.296} C_VEL
LIN {X 0,Y 335.244,Z 999.843,A -85,B 0,C 180,E1 13008.852,E2 13008.852} C_VEL
LIN {X 0,Y 331.322,Z 1024.189,A -85,B 0,C 180,E1 13007.679,E2 13007.679} C_VEL
LIN {X 0,Y 327.815,Z 1042.24,A -85,B 0,C 180,E1 13006.59,E2 13006.59} C_VEL
LIN {X 0,Y 325.494,Z 1049.325,A -85,B 0,C 180,E1 13006.208,E2 13006.208} C_VEL
LIN {X 0,Y 315.807,Z 1067.65,A -85,B 0,C 180,E1 13005.37,E2 13005.37} C_VEL
LIN {X 0,Y 313.622,Z 1073.45,A -85,B 0,C 180,E1 13004.925,E2 13004.925} C_VEL
LIN {X 0,Y 307.889,Z 1094.272,A -85,B 0,C 180,E1 13002.873,E2 13002.873} C_VEL
LIN {X 0,Y 301.379,Z 1115.553,A -85,B 0,C 180,E1 13000.313,E2 13000.313} C_VEL
LIN {X 0,Y 295.092,Z 1134.591,A -85,B 0,C 180,E1 12997.541,E2 12997.541} C_VEL
LIN {X 0,Y 289.059,Z 1152.095,A -85,B 0,C 180,E1 12994.492,E2 12994.492} C_VEL
LIN {X 0,Y 283.203,Z 1168.736,A -85,B 0,C 180,E1 12991.029,E2 12991.029} C_VEL
LIN {X 0,Y 278.03,Z 1183.597,A -85,B 0,C 180,E1 12987.336,E2 12987.336} C_VEL
LIN {X 0,Y 273.467,Z 1197.254,A -85,B 0,C 180,E1 12983.259,E2 12983.259} C_VEL
LIN {X 0,Y 269.889,Z 1208.939,A -85,B 0,C 180,E1 12979.028,E2 12979.028} C_VEL
LIN {X 0,Y 267.206,Z 1219.24,A -85,B 0,C 180,E1 12974.52,E2 12974.52} C_VEL
LIN {X 0,Y 265.531,Z 1227.727,A -85,B 0,C 180,E1 12969.975,E2 12969.975} C_VEL
LIN {X 0,Y 264.692,Z 1234.174,A -85,B 0,C 180,E1 12965.637,E2 12965.637} C_VEL
LIN {X 0,Y 264.403,Z 1239.426,A -85,B 0,C 180,E1 12961.083,E2 12961.083} C_VEL
LIN {X 0,Y 264.44,Z 1243.136,A -85,B 0,C 180,E1 12956.749,E2 12956.749} C_VEL
LIN {X 0,Y 264.823,Z 1245.667,A -85,B 0,C 180,E1 12952.188,E2 12952.188} C_VEL
LIN {X 0,Y 265.909,Z 1247.104,A -85,B 0,C 180,E1 12947.182,E2 12947.182} C_VEL
LIN {X 0,Y 268.404,Z 1247.021,A -85,B 0,C 180,E1 12941.764,E2 12941.764} C_VEL
LIN {X 0,Y 273.087,Z 1245.115,A -85,B 0,C 180,E1 12936.02,E2 12936.02} C_VEL
LIN {X 0,Y 280.425,Z 1241.228,A -85,B 0,C 180,E1 12930.289,E2 12930.289} C_VEL
LIN {X 0,Y 290.387,Z 1235.415,A -85,B 0,C 180,E1 12924.898,E2 12924.898} C_VEL
LIN {X 0,Y 302.647,Z 1227.922,A -85,B 0,C 180,E1 12920.042,E2 12920.042} C_VEL
LIN {X 0,Y 317.447,Z 1218.619,A -85,B 0,C 180,E1 12915.633,E2 12915.633} C_VEL
LIN {X 0,Y 321.583,Z 1216.058,A -85,B 0,C 180,E1 12914.561,E2 12914.561} C_VEL
LIN {X 0,Y 304.646,Z 1228.256,A -85,B 0,C 180,E1 12910.534,E2 12910.534} C_VEL
LIN {X 0,Y 289.217,Z 1241.335,A -85,B 0,C 180,E1 12905.268,E2 12905.268} C_VEL
LIN {X 0,Y 277.785,Z 1252.874,A -85,B 0,C 180,E1 12899.415,E2 12899.415} C_VEL
LIN {X 0,Y 270.681,Z 1261.509,A -85,B 0,C 180,E1 12893.746,E2 12893.746} C_VEL
LIN {X 0,Y 266.54,Z 1267.75,A -85,B 0,C 180,E1 12888.144,E2 12888.144} C_VEL
LIN {X 0,Y 264.723,Z 1271.45,A -85,B 0,C 180,E1 12883.101,E2 12883.101} C_VEL
LIN {X 0,Y 264.262,Z 1273.186,A -85,B 0,C 180,E1 12878.489,E2 12878.489} C_VEL
LIN {X 0,Y 264.473,Z 1273.273,A -85,B 0,C 180,E1 12874.122,E2 12874.122} C_VEL
LIN {X 0,Y 264.769,Z 1271.949,A -85,B 0,C 180,E1 12870.219,E2 12870.219} C_VEL
LIN {X 0,Y 264.821,Z 1269.388,A -85,B 0,C 180,E1 12866.54,E2 12866.54} C_VEL
LIN {X 0,Y 264.754,Z 1265.173,A -85,B 0,C 180,E1 12862.626,E2 12862.626} C_VEL
LIN {X 0,Y 264.884,Z 1259.05,A -85,B 0,C 180,E1 12858.462,E2 12858.462} C_VEL
LIN {X 0,Y 265.595,Z 1250.693,A -85,B 0,C 180,E1 12854.052,E2 12854.052} C_VEL
LIN {X 0,Y 267.244,Z 1239.793,A -85,B 0,C 180,E1 12849.412,E2 12849.412} C_VEL
LIN {X 0,Y 269.881,Z 1227.237,A -85,B 0,C 180,E1 12845.02,E2 12845.02} C_VEL
LIN {X 0,Y 273.674,Z 1212.466,A -85,B 0,C 180,E1 12840.691,E2 12840.691} C_VEL
LIN {X 0,Y 278.705,Z 1195.258,A -85,B 0,C 180,E1 12836.466,E2 12836.466} C_VEL
LIN {X 0,Y 284.684,Z 1176.501,A -85,B 0,C 180,E1 12832.586,E2 12832.586} C_VEL
LIN {X 0,Y 291.836,Z 1155.118,A -85,B 0,C 180,E1 12828.87,E2 12828.87} C_VEL
LIN {X 0,Y 299.927,Z 1131.394,A -85,B 0,C 180,E1 12825.436,E2 12825.436} C_VEL
LIN {X 0,Y 309.448,Z 1103.569,A -85,B 0,C 180,E1 12822.14,E2 12822.14} C_VEL
LIN {X 0,Y 318.389,Z 1077.369,A -85,B 0,C 180,E1 12819.563,E2 12819.563} C_VEL
LIN {X 0,Y 327.27,Z 1050.519,A -85,B 0,C 180,E1 12817.41,E2 12817.41} C_VEL
LIN {X 0,Y 336.168,Z 1022.307,A -85,B 0,C 180,E1 12815.567,E2 12815.567} C_VEL
LIN {X 0,Y 343.14,Z 997.716,A -85,B 0,C 180,E1 12814.221,E2 12814.221} C_VEL
LIN {X 0,Y 338.742,Z 972.794,A -85,B 0,C 180,E1 12811.597,E2 12811.597} C_VEL
LIN {X 0,Y 335.853,Z 948.811,A -85,B 0,C 180,E1 12809.361,E2 12809.361} C_VEL
LIN {X 0,Y 333.914,Z 924.452,A -85,B 0,C 180,E1 12807.377,E2 12807.377} C_VEL
LIN {X 0,Y 332.973,Z 896.736,A -85,B 0,C 180,E1 12805.407,E2 12805.407} C_VEL
LIN {X 0,Y 333.208,Z 881.159,A -85,B 0,C 180,E1 12804.369,E2 12804.369} C_VEL
LIN {X 0,Y 343.257,Z 847.668,A -85,B 0,C 180,E1 12800.202,E2 12800.202} C_VEL
LIN {X 0,Y 348.296,Z 831.277,A -85,B 0,C 180,E1 12798.161,E2 12798.161} C_VEL
LIN {X 0,Y 342.768,Z 815.12,A -85,B 0,C 180,E1 12794.184,E2 12794.184} C_VEL
LIN {X 0,Y 337.032,Z 799.494,A -85,B 0,C 180,E1 12789.967,E2 12789.967} C_VEL
LIN {X 0,Y 331.685,Z 785.627,A -85,B 0,C 180,E1 12785.871,E2 12785.871} C_VEL
LIN {X 0,Y 326.753,Z 773.501,A -85,B 0,C 180,E1 12781.929,E2 12781.929} C_VEL
LIN {X 0,Y 322.347,Z 763.041,A -85,B 0,C 180,E1 12778.222,E2 12778.222} C_VEL
LIN {X 0,Y 317.916,Z 752.689,A -85,B 0,C 180,E1 12774.224,E2 12774.224} C_VEL
LIN {X 0,Y 312.826,Z 741.283,A -85,B 0,C 180,E1 12769.316,E2 12769.316} C_VEL
LIN {X 0,Y 308.566,Z 732.134,A -85,B 0,C 180,E1 12764.927,E2 12764.927} C_VEL
LIN {X 0,Y 305.552,Z 725.946,A -85,B 0,C 180,E1 12761.611,E2 12761.611} C_VEL
LIN {X 0,Y 302.53,Z 719.381,A -85,B 0,C 180,E1 12757.865,E2 12757.865} C_VEL
LIN {X 0,Y 299.903,Z 714.215,A -85,B 0,C 180,E1 12754.526,E2 12754.526} C_VEL
LIN {X 0,Y 298.009,Z 710.197,A -85,B 0,C 180,E1 12751.765,E2 12751.765} C_VEL
LIN {X 0,Y 297.818,Z 709.809,A -85,B 0,C 180,E1 12751.362,E2 12751.362} C_VEL
LIN {X 0,Y 302.159,Z 711.007,A -85,B 0,C 180,E1 12749.802,E2 12749.802} C_VEL
LIN {X 0,Y 307.765,Z 723.969,A -85,B 0,C 180,E1 12746.251,E2 12746.251} C_VEL
LIN {X 0,Y 313.329,Z 738.57,A -85,B 0,C 180,E1 12742.905,E2 12742.905} C_VEL
LIN {X 0,Y 317.808,Z 752.736,A -85,B 0,C 180,E1 12740.072,E2 12740.072} C_VEL
LIN {X 0,Y 320.988,Z 764.838,A -85,B 0,C 180,E1 12737.899,E2 12737.899} C_VEL
LIN {X 0,Y 314.102,Z 812.273,A -85,B 0,C 180,E1 12733.436,E2 12733.436} C_VEL
LIN {X 0,Y 307.587,Z 861.408,A -85,B 0,C 180,E1 12728.854,E2 12728.854} C_VEL
LIN {X 0,Y 305.702,Z 877.883,A -85,B 0,C 180,E1 12727.373,E2 12727.373} C_VEL
LIN {X 0,Y 305.934,Z 884.466,A -85,B 0,C 180,E1 12727.144,E2 12727.144} C_VEL
LIN {X 0,Y 298.827,Z 1034.27,A -85,B 0,C 180,E1 12723.792,E2 12723.792} C_VEL
LIN {X 0,Y 298.083,Z 1054.711,A -85,B 0,C 180,E1 12723.163,E2 12723.163} C_VEL
LIN {X 0,Y 296.674,Z 1072.15,A -85,B 0,C 180,E1 12722.293,E2 12722.293} C_VEL
LIN {X 0,Y 294.644,Z 1088.199,A -85,B 0,C 180,E1 12721.162,E2 12721.162} C_VEL
LIN {X 0,Y 291.909,Z 1104.141,A -85,B 0,C 180,E1 12719.664,E2 12719.664} C_VEL
LIN {X 0,Y 288.759,Z 1119.037,A -85,B 0,C 180,E1 12717.867,E2 12717.867} C_VEL
LIN {X 0,Y 285.27,Z 1133.032,A -85,B 0,C 180,E1 12715.736,E2 12715.736} C_VEL
LIN {X 0,Y 281.822,Z 1145.169,A -85,B 0,C 180,E1 12713.41,E2 12713.41} C_VEL
LIN {X 0,Y 278.187,Z 1156.771,A -85,B 0,C 180,E1 12710.621,E2 12710.621} C_VEL
LIN {X 0,Y 274.855,Z 1166.784,A -85,B 0,C 180,E1 12707.571,E2 12707.571} C_VEL
LIN {X 0,Y 272.115,Z 1174.738,A -85,B 0,C 180,E1 12704.466,E2 12704.466} C_VEL
LIN {X 0,Y 269.845,Z 1181.255,A -85,B 0,C 180,E1 12701.106,E2 12701.106} C_VEL
LIN {X 0,Y 268.149,Z 1186.284,A -85,B 0,C 180,E1 12697.496,E2 12697.496} C_VEL
LIN {X 0,Y 267.125,Z 1189.557,A -85,B 0,C 180,E1 12693.86,E2 12693.86} C_VEL
LIN {X 0,Y 266.692,Z 1191.224,A -85,B 0,C 180,E1 12689.997,E2 12689.997} C_VEL
LIN {X 0,Y 266.855,Z 1191.035,A -85,B 0,C 180,E1 12686.13,E2 12686.13} C_VEL
LIN {X 0,Y 267.658,Z 1189.065,A -85,B 0,C 180,E1 12682.268,E2 12682.268} C_VEL
LIN {X 0,Y 269.088,Z 1185.481,A -85,B 0,C 180,E1 12678.639,E2 12678.639} C_VEL
LIN {X 0,Y 271.224,Z 1180.019,A -85,B 0,C 180,E1 12675.042,E2 12675.042} C_VEL
LIN {X 0,Y 274.136,Z 1172.546,A -85,B 0,C 180,E1 12671.496,E2 12671.496} C_VEL
LIN {X 0,Y 277.362,Z 1164.022,A -85,B 0,C 180,E1 12668.423,E2 12668.423} C_VEL
LIN {X 0,Y 280.911,Z 1154.058,A -85,B 0,C 180,E1 12665.61,E2 12665.61} C_VEL
LIN {X 0,Y 284.64,Z 1142.636,A -85,B 0,C 180,E1 12663.051,E2 12663.051} C_VEL
LIN {X 0,Y 288.599,Z 1129.118,A -85,B 0,C 180,E1 12660.641,E2 12660.641} C_VEL
LIN {X 0,Y 292.176,Z 1115.061,A -85,B 0,C 180,E1 12658.653,E2 12658.653} C_VEL
LIN {X 0,Y 295.364,Z 1099.862,A -85,B 0,C 180,E1 12656.971,E2 12656.971} C_VEL
LIN {X 0,Y 298.059,Z 1083.54,A -85,B 0,C 180,E1 12655.577,E2 12655.577} C_VEL
LIN {X 0,Y 300.092,Z 1066.482,A -85,B 0,C 180,E1 12654.498,E2 12654.498} C_VEL
LIN {X 0,Y 301.293,Z 1048.942,A -85,B 0,C 180,E1 12653.75,E2 12653.75} C_VEL
LIN {X 0,Y 302.992,Z 1005.03,A -85,B 0,C 180,E1 12652.639,E2 12652.639} C_VEL
LIN {X 0,Y 304.574,Z 1005.865,A -85,B 0,C 180,E1 12652.363,E2 12652.363} C_VEL
LIN {X 0,Y 306.85,Z 1004.817,A -85,B 0,C 180,E1 12652.13,E2 12652.13} C_VEL
LIN {X 0,Y 310.059,Z 1000.768,A -85,B 0,C 180,E1 12651.977,E2 12651.977} C_VEL
LIN {X 0,Y 313.909,Z 992.478,A -85,B 0,C 180,E1 12651.996,E2 12651.996} C_VEL
LIN {X 0,Y 314.754,Z 990.559,A -85,B 0,C 180,E1 12652.004,E2 12652.004} C_VEL
LIN {X 0,Y 318.612,Z 987.441,A -85,B 0,C 180,E1 12651.681,E2 12651.681} C_VEL
LIN {X 0,Y 322.617,Z 981.761,A -85,B 0,C 180,E1 12651.493,E2 12651.493} C_VEL
LIN {X 0,Y 327.132,Z 972.306,A -85,B 0,C 180,E1 12651.456,E2 12651.456} C_VEL
LIN {X 0,Y 331.692,Z 967.338,A -85,B 0,C 180,E1 12651.139,E2 12651.139} C_VEL
LIN {X 0,Y 333.8,Z 964.33,A -85,B 0,C 180,E1 12651.034,E2 12651.034} C_VEL
LIN {X 0,Y 327.354,Z 1008.889,A -85,B 0,C 180,E1 12649.245,E2 12649.245} C_VEL
LIN {X 0,Y 323.08,Z 1032.603,A -85,B 0,C 180,E1 12647.968,E2 12647.968} C_VEL
LIN {X 0,Y 318.227,Z 1054.91,A -85,B 0,C 180,E1 12646.45,E2 12646.45} C_VEL
LIN {X 0,Y 313.622,Z 1073.45,A -85,B 0,C 180,E1 12644.925,E2 12644.925} C_VEL
LIN {X 0,Y 310.943,Z 1080.274,A -85,B 0,C 180,E1 12644.388,E2 12644.388} C_VEL
LIN {X 0,Y 300.534,Z 1097.547,A -85,B 0,C 180,E1 12643.154,E2 12643.154} C_VEL
LIN {X 0,Y 298.207,Z 1102.938,A -85,B 0,C 180,E1 12642.589,E2 12642.589} C_VEL
LIN {X 0,Y 291.787,Z 1122.799,A -85,B 0,C 180,E1 12639.98,E2 12639.98} C_VEL
LIN {X 0,Y 285.181,Z 1142.059,A -85,B 0,C 180,E1 12636.923,E2 12636.923} C_VEL
LIN {X 0,Y 279.177,Z 1158.895,A -85,B 0,C 180,E1 12633.721,E2 12633.721} C_VEL
LIN {X 0,Y 273.404,Z 1174.94,A -85,B 0,C 180,E1 12630.069,E2 12630.069} C_VEL
LIN {X 0,Y 268.226,Z 1189.569,A -85,B 0,C 180,E1 12626.047,E2 12626.047} C_VEL
LIN {X 0,Y 263.961,Z 1202.432,A -85,B 0,C 180,E1 12621.791,E2 12621.791} C_VEL
LIN {X 0,Y 260.576,Z 1214.007,A -85,B 0,C 180,E1 12617.155,E2 12617.155} C_VEL
LIN {X 0,Y 258.326,Z 1223.506,A -85,B 0,C 180,E1 12612.519,E2 12612.519} C_VEL
LIN {X 0,Y 257.067,Z 1230.901,A -85,B 0,C 180,E1 12608.049,E2 12608.049} C_VEL
LIN {X 0,Y 256.486,Z 1237.065,A -85,B 0,C 180,E1 12603.352,E2 12603.352} C_VEL
LIN {X 0,Y 256.389,Z 1241.6,A -85,B 0,C 180,E1 12598.883,E2 12598.883} C_VEL
LIN {X 0,Y 256.606,Z 1244.918,A -85,B 0,C 180,E1 12594.185,E2 12594.185} C_VEL
LIN {X 0,Y 257.353,Z 1247.138,A -85,B 0,C 180,E1 12589.252,E2 12589.252} C_VEL
LIN {X 0,Y 259.257,Z 1248.008,A -85,B 0,C 180,E1 12583.816,E2 12583.816} C_VEL
LIN {X 0,Y 263.032,Z 1247.271,A -85,B 0,C 180,E1 12578.128,E2 12578.128} C_VEL
LIN {X 0,Y 269.02,Z 1244.882,A -85,B 0,C 180,E1 12572.556,E2 12572.556} C_VEL
LIN {X 0,Y 277.832,Z 1240.639,A -85,B 0,C 180,E1 12566.99,E2 12566.99} C_VEL
LIN {X 0,Y 289.346,Z 1234.612,A -85,B 0,C 180,E1 12561.788,E2 12561.788} C_VEL
LIN {X 0,Y 303.611,Z 1226.784,A -85,B 0,C 180,E1 12557.022,E2 12557.022} C_VEL
LIN {X 0,Y 312.253,Z 1221.931,A -85,B 0,C 180,E1 12554.661,E2 12554.661} C_VEL
LIN {X 0,Y 295.512,Z 1233.224,A -85,B 0,C 180,E1 12550.518,E2 12550.518} C_VEL
LIN {X 0,Y 280.2,Z 1245.281,A -85,B 0,C 180,E1 12545.069,E2 12545.069} C_VEL
LIN {X 0,Y 269.078,Z 1255.583,A -85,B 0,C 180,E1 12539.133,E2 12539.133} C_VEL
LIN {X 0,Y 262.192,Z 1263.185,A -85,B 0,C 180,E1 12533.369,E2 12533.369} C_VEL
LIN {X 0,Y 258.318,Z 1268.428,A -85,B 0,C 180,E1 12527.809,E2 12527.809} C_VEL
LIN {X 0,Y 256.619,Z 1271.509,A -85,B 0,C 180,E1 12522.606,E2 12522.606} C_VEL
LIN {X 0,Y 256.287,Z 1272.712,A -85,B 0,C 180,E1 12517.705,E2 12517.705} C_VEL
LIN {X 0,Y 256.557,Z 1272.361,A -85,B 0,C 180,E1 12513.578,E2 12513.578} C_VEL
LIN {X 0,Y 256.848,Z 1270.727,A -85,B 0,C 180,E1 12509.78,E2 12509.78} C_VEL
LIN {X 0,Y 256.882,Z 1267.807,A -85,B 0,C 180,E1 12505.985,E2 12505.985} C_VEL
LIN {X 0,Y 256.818,Z 1263.24,A -85,B 0,C 180,E1 12501.946,E2 12501.946} C_VEL
LIN {X 0,Y 257.028,Z 1256.544,A -85,B 0,C 180,E1 12497.539,E2 12497.539} C_VEL
LIN {X 0,Y 257.871,Z 1247.97,A -85,B 0,C 180,E1 12493.097,E2 12493.097} C_VEL
LIN {X 0,Y 259.665,Z 1237.162,A -85,B 0,C 180,E1 12488.546,E2 12488.546} C_VEL
LIN {X 0,Y 262.73,Z 1223.516,A -85,B 0,C 180,E1 12483.806,E2 12483.806} C_VEL
LIN {X 0,Y 266.902,Z 1208.177,A -85,B 0,C 180,E1 12479.374,E2 12479.374} C_VEL
LIN {X 0,Y 272.215,Z 1190.913,A -85,B 0,C 180,E1 12475.172,E2 12475.172} C_VEL
LIN {X 0,Y 279.151,Z 1169.97,A -85,B 0,C 180,E1 12470.924,E2 12470.924} C_VEL
LIN {X 0,Y 287.274,Z 1146.451,A -85,B 0,C 180,E1 12466.989,E2 12466.989} C_VEL
LIN {X 0,Y 296.038,Z 1121.473,A -85,B 0,C 180,E1 12463.553,E2 12463.553} C_VEL
LIN {X 0,Y 305.288,Z 1094.992,A -85,B 0,C 180,E1 12460.553,E2 12460.553} C_VEL
LIN {X 0,Y 314.709,Z 1067.771,A -85,B 0,C 180,E1 12458.011,E2 12458.011} C_VEL
LIN {X 0,Y 323.968,Z 1040.084,A -85,B 0,C 180,E1 12455.892,E2 12455.892} C_VEL
LIN {X 0,Y 332.992,Z 1011.683,A -85,B 0,C 180,E1 12454.144,E2 12454.144} C_VEL
LIN {X 0,Y 336.404,Z 999.708,A -85,B 0,C 180,E1 12453.512,E2 12453.512} C_VEL
LIN {X 0,Y 332.297,Z 974.308,A -85,B 0,C 180,E1 12450.766,E2 12450.766} C_VEL
LIN {X 0,Y 329.502,Z 948.465,A -85,B 0,C 180,E1 12448.321,E2 12448.321} C_VEL
LIN {X 0,Y 327.897,Z 922.971,A -85,B 0,C 180,E1 12446.218,E2 12446.218} C_VEL
LIN {X 0,Y 327.342,Z 894.019,A -85,B 0,C 180,E1 12444.174,E2 12444.174} C_VEL
LIN {X 0,Y 327.703,Z 879.184,A -85,B 0,C 180,E1 12443.179,E2 12443.179} C_VEL
LIN {X 0,Y 337.732,Z 846.782,A -85,B 0,C 180,E1 12439.105,E2 12439.105} C_VEL
LIN {X 0,Y 341.541,Z 834.495,A -85,B 0,C 180,E1 12437.55,E2 12437.55} C_VEL
LIN {X 0,Y 336.145,Z 818.688,A -85,B 0,C 180,E1 12433.591,E2 12433.591} C_VEL
LIN {X 0,Y 330.577,Z 803.424,A -85,B 0,C 180,E1 12429.4,E2 12429.4} C_VEL
LIN {X 0,Y 325.582,Z 790.333,A -85,B 0,C 180,E1 12425.463,E2 12425.463} C_VEL
LIN {X 0,Y 320.469,Z 777.604,A -85,B 0,C 180,E1 12421.251,E2 12421.251} C_VEL
LIN {X 0,Y 315.43,Z 765.488,A -85,B 0,C 180,E1 12416.827,E2 12416.827} C_VEL
LIN {X 0,Y 310.666,Z 754.507,A -85,B 0,C 180,E1 12412.415,E2 12412.415} C_VEL
LIN {X 0,Y 306.417,Z 745.139,A -85,B 0,C 180,E1 12408.207,E2 12408.207} C_VEL
LIN {X 0,Y 302.98,Z 737.563,A -85,B 0,C 180,E1 12404.492,E2 12404.492} C_VEL
LIN {X 0,Y 299.601,Z 730.132,A -85,B 0,C 180,E1 12400.504,E2 12400.504} C_VEL
LIN {X 0,Y 296.666,Z 724.279,A -85,B 0,C 180,E1 12396.936,E2 12396.936} C_VEL
LIN {X 0,Y 294.67,Z 720.137,A -85,B 0,C 180,E1 12394.257,E2 12394.257} C_VEL
LIN {X 0,Y 293.146,Z 716.604,A -85,B 0,C 180,E1 12391.809,E2 12391.809} C_VEL
LIN {X 0,Y 298.133,Z 718.308,A -85,B 0,C 180,E1 12389.909,E2 12389.909} C_VEL
LIN {X 0,Y 303.269,Z 730.705,A -85,B 0,C 180,E1 12386.522,E2 12386.522} C_VEL
LIN {X 0,Y 308.289,Z 744.32,A -85,B 0,C 180,E1 12383.36,E2 12383.36} C_VEL
LIN {X 0,Y 312.672,Z 758.879,A -85,B 0,C 180,E1 12380.411,E2 12380.411} C_VEL
LIN {X 0,Y 314.959,Z 768.45,A -85,B 0,C 180,E1 12378.675,E2 12378.675} C_VEL
LIN {X 0,Y 307.661,Z 817.181,A -85,B 0,C 180,E1 12374.062,E2 12374.062} C_VEL
LIN {X 0,Y 300.706,Z 867.695,A -85,B 0,C 180,E1 12369.3,E2 12369.3} C_VEL
LIN {X 0,Y 299.463,Z 878.993,A -85,B 0,C 180,E1 12368.301,E2 12368.301} C_VEL
LIN {X 0,Y 299.66,Z 885.387,A -85,B 0,C 180,E1 12368.075,E2 12368.075} C_VEL
LIN {X 0,Y 292.3,Z 1034.636,A -85,B 0,C 180,E1 12364.686,E2 12364.686} C_VEL
LIN {X 0,Y 291.513,Z 1055.39,A -85,B 0,C 180,E1 12364.041,E2 12364.041} C_VEL
LIN {X 0,Y 290.043,Z 1072.921,A -85,B 0,C 180,E1 12363.154,E2 12363.154} C_VEL
LIN {X 0,Y 287.887,Z 1089.307,A -85,B 0,C 180,E1 12361.979,E2 12361.979} C_VEL
LIN {X 0,Y 285.045,Z 1105.217,A -85,B 0,C 180,E1 12360.453,E2 12360.453} C_VEL
LIN {X 0,Y 281.648,Z 1120.617,A -85,B 0,C 180,E1 12358.548,E2 12358.548} C_VEL
LIN {X 0,Y 278.021,Z 1134.516,A -85,B 0,C 180,E1 12356.366,E2 12356.366} C_VEL
LIN {X 0,Y 274.269,Z 1147.084,A -85,B 0,C 180,E1 12353.867,E2 12353.867} C_VEL
LIN {X 0,Y 270.523,Z 1158.525,A -85,B 0,C 180,E1 12351.006,E2 12351.006} C_VEL
LIN {X 0,Y 267.089,Z 1168.391,A -85,B 0,C 180,E1 12347.874,E2 12347.874} C_VEL
LIN {X 0,Y 264.094,Z 1176.613,A -85,B 0,C 180,E1 12344.467,E2 12344.467} C_VEL
LIN {X 0,Y 261.688,Z 1183.254,A -85,B 0,C 180,E1 12340.788,E2 12340.788} C_VEL
LIN {X 0,Y 260.041,Z 1187.988,A -85,B 0,C 180,E1 12337.065,E2 12337.065} C_VEL
LIN {X 0,Y 259.08,Z 1190.931,A -85,B 0,C 180,E1 12333.316,E2 12333.316} C_VEL
LIN {X 0,Y 258.731,Z 1192.247,A -85,B 0,C 180,E1 12329.333,E2 12329.333} C_VEL
LIN {X 0,Y 259.021,Z 1191.792,A -85,B 0,C 180,E1 12325.347,E2 12325.347} C_VEL
LIN {X 0,Y 259.922,Z 1189.698,A -85,B 0,C 180,E1 12321.591,E2 12321.591} C_VEL
LIN {X 0,Y 261.509,Z 1185.846,A -85,B 0,C 180,E1 12317.858,E2 12317.858} C_VEL
LIN {X 0,Y 263.855,Z 1180.163,A -85,B 0,C 180,E1 12314.163,E2 12314.163} C_VEL
LIN {X 0,Y 266.803,Z 1172.963,A -85,B 0,C 180,E1 12310.741,E2 12310.741} C_VEL
LIN {X 0,Y 270.221,Z 1164.286,A -85,B 0,C 180,E1 12307.594,E2 12307.594} C_VEL
LIN {X 0,Y 273.961,Z 1154.124,A -85,B 0,C 180,E1 12304.719,E2 12304.719} C_VEL
LIN {X 0,Y 277.883,Z 1142.523,A -85,B 0,C 180,E1 12302.108,E2 12302.108} C_VEL
LIN {X 0,Y 281.864,Z 1129.378,A -85,B 0,C 180,E1 12299.75,E2 12299.75} C_VEL
LIN {X 0,Y 285.407,Z 1115.88,A -85,B 0,C 180,E1 12297.822,E2 12297.822} C_VEL
LIN {X 0,Y 288.721,Z 1100.642,A -85,B 0,C 180,E1 12296.109,E2 12296.109} C_VEL
LIN {X 0,Y 291.522,Z 1084.269,A -85,B 0,C 180,E1 12294.692,E2 12294.692} C_VEL
LIN {X 0,Y 293.625,Z 1067.221,A -85,B 0,C 180,E1 12293.6,E2 12293.6} C_VEL
LIN {X 0,Y 294.87,Z 1049.658,A -85,B 0,C 180,E1 12292.843,E2 12292.843} C_VEL
LIN {X 0,Y 295.772,Z 1024.006,A -85,B 0,C 180,E1 12292.148,E2 12292.148} C_VEL
LIN {X 0,Y 297.679,Z 1024.767,A -85,B 0,C 180,E1 12291.824,E2 12291.824} C_VEL
LIN {X 0,Y 299.744,Z 1023.859,A -85,B 0,C 180,E1 12291.621,E2 12291.621} C_VEL
LIN {X 0,Y 302.876,Z 1020.474,A -85,B 0,C 180,E1 12291.482,E2 12291.482} C_VEL
LIN {X 0,Y 306.497,Z 1013.871,A -85,B 0,C 180,E1 12291.532,E2 12291.532} C_VEL
LIN {X 0,Y 307.14,Z 1012.554,A -85,B 0,C 180,E1 12291.55,E2 12291.55} C_VEL
LIN {X 0,Y 311.008,Z 1009.75,A -85,B 0,C 180,E1 12291.233,E2 12291.233} C_VEL
LIN {X 0,Y 315.029,Z 1004.576,A -85,B 0,C 180,E1 12291.062,E2 12291.062} C_VEL
LIN {X 0,Y 319.248,Z 995.982,A -85,B 0,C 180,E1 12291.074,E2 12291.074} C_VEL
LIN {X 0,Y 323.35,Z 991.911,A -85,B 0,C 180,E1 12290.789,E2 12290.789} C_VEL
LIN {X 0,Y 319.28,Z 1017.398,A -85,B 0,C 180,E1 12289.622,E2 12289.622} C_VEL
LIN {X 0,Y 314.818,Z 1040.111,A -85,B 0,C 180,E1 12288.278,E2 12288.278} C_VEL
LIN {X 0,Y 309.555,Z 1062.594,A -85,B 0,C 180,E1 12286.617,E2 12286.617} C_VEL
LIN {X 0,Y 303.83,Z 1084.099,A -85,B 0,C 180,E1 12284.662,E2 12284.662} C_VEL
LIN {X 0,Y 298.207,Z 1102.938,A -85,B 0,C 180,E1 12282.589,E2 12282.589} C_VEL
LIN {X 0,Y 295.366,Z 1109.263,A -85,B 0,C 180,E1 12281.91,E2 12281.91} C_VEL
LIN {X 0,Y 284.432,Z 1125.39,A -85,B 0,C 180,E1 12280.235,E2 12280.235} C_VEL
LIN {X 0,Y 281.958,Z 1130.434,A -85,B 0,C 180,E1 12279.51,E2 12279.51} C_VEL
LIN {X 0,Y 275.321,Z 1148.989,A -85,B 0,C 180,E1 12276.297,E2 12276.297} C_VEL
LIN {X 0,Y 268.891,Z 1166.439,A -85,B 0,C 180,E1 12272.629,E2 12272.629} C_VEL
LIN {X 0,Y 263.364,Z 1181.432,A -85,B 0,C 180,E1 12268.827,E2 12268.827} C_VEL
LIN {X 0,Y 258.436,Z 1195.357,A -85,B 0,C 180,E1 12264.597,E2 12264.597} C_VEL
LIN {X 0,Y 254.457,Z 1207.685,A -85,B 0,C 180,E1 12260.084,E2 12260.084} C_VEL
LIN {X 0,Y 251.568,Z 1218.177,A -85,B 0,C 180,E1 12255.444,E2 12255.444} C_VEL
LIN {X 0,Y 249.677,Z 1226.996,A -85,B 0,C 180,E1 12250.616,E2 12250.616} C_VEL
LIN {X 0,Y 248.703,Z 1234.137,A -85,B 0,C 180,E1 12245.769,E2 12245.769} C_VEL
LIN {X 0,Y 248.404,Z 1239.522,A -85,B 0,C 180,E1 12241.153,E2 12241.153} C_VEL
LIN {X 0,Y 248.456,Z 1243.553,A -85,B 0,C 180,E1 12236.464,E2 12236.464} C_VEL
LIN {X 0,Y 248.939,Z 1246.605,A -85,B 0,C 180,E1 12231.453,E2 12231.453} C_VEL
LIN {X 0,Y 250.261,Z 1248.338,A -85,B 0,C 180,E1 12226.13,E2 12226.13} C_VEL
LIN {X 0,Y 253.238,Z 1248.704,A -85,B 0,C 180,E1 12220.39,E2 12220.39} C_VEL
LIN {X 0,Y 258.696,Z 1247.385,A -85,B 0,C 180,E1 12214.349,E2 12214.349} C_VEL
LIN {X 0,Y 267.051,Z 1244.219,A -85,B 0,C 180,E1 12208.386,E2 12208.386} C_VEL
LIN {X 0,Y 278.647,Z 1239.086,A -85,B 0,C 180,E1 12202.668,E2 12202.668} C_VEL
LIN {X 0,Y 292.582,Z 1232.425,A -85,B 0,C 180,E1 12197.682,E2 12197.682} C_VEL
LIN {X 0,Y 302.894,Z 1227.312,A -85,B 0,C 180,E1 12194.786,E2 12194.786} C_VEL
LIN {X 0,Y 284.694,Z 1238.862,A -85,B 0,C 180,E1 12189.998,E2 12189.998} C_VEL
LIN {X 0,Y 269.87,Z 1249.797,A -85,B 0,C 180,E1 12184.278,E2 12184.278} C_VEL
LIN {X 0,Y 259.586,Z 1258.65,A -85,B 0,C 180,E1 12178.283,E2 12178.283} C_VEL
LIN {X 0,Y 253.318,Z 1264.993,A -85,B 0,C 180,E1 12172.515,E2 12172.515} C_VEL
LIN {X 0,Y 249.891,Z 1269.192,A -85,B 0,C 180,E1 12166.986,E2 12166.986} C_VEL
LIN {X 0,Y 248.472,Z 1271.507,A -85,B 0,C 180,E1 12161.611,E2 12161.611} C_VEL
LIN {X 0,Y 248.366,Z 1272.017,A -85,B 0,C 180,E1 12156.708,E2 12156.708} C_VEL
LIN {X 0,Y 248.704,Z 1271.087,A -85,B 0,C 180,E1 12152.538,E2 12152.538} C_VEL
LIN {X 0,Y 248.95,Z 1268.921,A -85,B 0,C 180,E1 12148.622,E2 12148.622} C_VEL
LIN {X 0,Y 248.931,Z 1265.449,A -85,B 0,C 180,E1 12144.702,E2 12144.702} C_VEL
LIN {X 0,Y 248.895,Z 1260.25,A -85,B 0,C 180,E1 12140.523,E2 12140.523} C_VEL
LIN {X 0,Y 249.266,Z 1253.041,A -85,B 0,C 180,E1 12136.077,E2 12136.077} C_VEL
LIN {X 0,Y 250.438,Z 1243.52,A -85,B 0,C 180,E1 12131.377,E2 12131.377} C_VEL
LIN {X 0,Y 252.661,Z 1231.919,A -85,B 0,C 180,E1 12126.691,E2 12126.691} C_VEL
LIN {X 0,Y 256.285,Z 1217.382,A -85,B 0,C 180,E1 12121.835,E2 12121.835} C_VEL
LIN {X 0,Y 260.857,Z 1201.801,A -85,B 0,C 180,E1 12117.489,E2 12117.489} C_VEL
LIN {X 0,Y 266.841,Z 1183.365,A -85,B 0,C 180,E1 12113.167,E2 12113.167} C_VEL
LIN {X 0,Y 274.258,Z 1161.906,A -85,B 0,C 180,E1 12108.99,E2 12108.99} C_VEL
LIN {X 0,Y 282.819,Z 1137.967,A -85,B 0,C 180,E1 12105.149,E2 12105.149} C_VEL
LIN {X 0,Y 291.591,Z 1113.443,A -85,B 0,C 180,E1 12101.922,E2 12101.922} C_VEL
LIN {X 0,Y 301.105,Z 1086.919,A -85,B 0,C 180,E1 12099.014,E2 12099.014} C_VEL
LIN {X 0,Y 310.896,Z 1059.139,A -85,B 0,C 180,E1 12096.512,E2 12096.512} C_VEL
LIN {X 0,Y 320.28,Z 1031.285,A -85,B 0,C 180,E1 12094.499,E2 12094.499} C_VEL
LIN {X 0,Y 329.452,Z 1001.964,A -85,B 0,C 180,E1 12092.792,E2 12092.792} C_VEL
LIN {X 0,Y 329.23,Z 999.327,A -85,B 0,C 180,E1 12092.518,E2 12092.518} C_VEL
LIN {X 0,Y 325.899,Z 976.521,A -85,B 0,C 180,E1 12090.007,E2 12090.007} C_VEL
LIN {X 0,Y 323.412,Z 950.113,A -85,B 0,C 180,E1 12087.43,E2 12087.43} C_VEL
LIN {X 0,Y 322.058,Z 924.698,A -85,B 0,C 180,E1 12085.295,E2 12085.295} C_VEL
LIN {X 0,Y 321.782,Z 895.916,A -85,B 0,C 180,E1 12083.215,E2 12083.215} C_VEL
LIN {X 0,Y 322.31,Z 877.109,A -85,B 0,C 180,E1 12081.949,E2 12081.949} C_VEL
LIN {X 0,Y 332.812,Z 844.097,A -85,B 0,C 180,E1 12077.762,E2 12077.762} C_VEL
LIN {X 0,Y 334.748,Z 837.704,A -85,B 0,C 180,E1 12076.932,E2 12076.932} C_VEL
LIN {X 0,Y 329.735,Z 822.861,A -85,B 0,C 180,E1 12073.146,E2 12073.146} C_VEL
LIN {X 0,Y 324.434,Z 808.149,A -85,B 0,C 180,E1 12069.043,E2 12069.043} C_VEL
LIN {X 0,Y 319.473,Z 795.005,A -85,B 0,C 180,E1 12065.028,E2 12065.028} C_VEL
LIN {X 0,Y 314.207,Z 781.679,A -85,B 0,C 180,E1 12060.547,E2 12060.547} C_VEL
LIN {X 0,Y 309.405,Z 770.224,A -85,B 0,C 180,E1 12056.294,E2 12056.294} C_VEL
LIN {X 0,Y 305.022,Z 759.914,A -85,B 0,C 180,E1 12052.086,E2 12052.086} C_VEL
LIN {X 0,Y 300.91,Z 750.743,A -85,B 0,C 180,E1 12047.916,E2 12047.916} C_VEL
LIN {X 0,Y 297.561,Z 743.273,A -85,B 0,C 180,E1 12044.206,E2 12044.206} C_VEL
LIN {X 0,Y 294.197,Z 735.797,A -85,B 0,C 180,E1 12040.131,E2 12040.131} C_VEL
LIN {X 0,Y 291.316,Z 729.975,A -85,B 0,C 180,E1 12036.537,E2 12036.537} C_VEL
LIN {X 0,Y 289.631,Z 726.378,A -85,B 0,C 180,E1 12034.215,E2 12034.215} C_VEL
LIN {X 0,Y 288.523,Z 723.597,A -85,B 0,C 180,E1 12032.217,E2 12032.217} C_VEL
LIN {X 0,Y 293.971,Z 725.298,A -85,B 0,C 180,E1 12030.113,E2 12030.113} C_VEL
LIN {X 0,Y 298.897,Z 737.717,A -85,B 0,C 180,E1 12026.727,E2 12026.727} C_VEL
LIN {X 0,Y 303.455,Z 750.911,A -85,B 0,C 180,E1 12023.622,E2 12023.622} C_VEL
LIN {X 0,Y 307.737,Z 765.987,A -85,B 0,C 180,E1 12020.564,E2 12020.564} C_VEL
LIN {X 0,Y 309.026,Z 772.036,A -85,B 0,C 180,E1 12019.492,E2 12019.492} C_VEL
LIN {X 0,Y 301.396,Z 820.84,A -85,B 0,C 180,E1 12014.823,E2 12014.823} C_VEL
LIN {X 0,Y 294.162,Z 872.081,A -85,B 0,C 180,E1 12009.969,E2 12009.969} C_VEL
LIN {X 0,Y 293.294,Z 879.942,A -85,B 0,C 180,E1 12009.276,E2 12009.276} C_VEL
LIN {X 0,Y 293.465,Z 886.353,A -85,B 0,C 180,E1 12009.046,E2 12009.046} C_VEL
LIN {X 0,Y 285.848,Z 1035.002,A -85,B 0,C 180,E1 12005.62,E2 12005.62} C_VEL
LIN {X 0,Y 285.014,Z 1056.072,A -85,B 0,C 180,E1 12004.959,E2 12004.959} C_VEL
LIN {X 0,Y 283.484,Z 1073.651,A -85,B 0,C 180,E1 12004.058,E2 12004.058} C_VEL
LIN {X 0,Y 281.376,Z 1089.266,A -85,B 0,C 180,E1 12002.932,E2 12002.932} C_VEL
LIN {X 0,Y 278.608,Z 1104.556,A -85,B 0,C 180,E1 12001.475,E2 12001.475} C_VEL
LIN {X 0,Y 275.186,Z 1119.727,A -85,B 0,C 180,E1 11999.61,E2 11999.61} C_VEL
LIN {X 0,Y 271.361,Z 1134.05,A -85,B 0,C 180,E1 11997.374,E2 11997.374} C_VEL
LIN {X 0,Y 267.636,Z 1146.303,A -85,B 0,C 180,E1 11994.968,E2 11994.968} C_VEL
LIN {X 0,Y 263.924,Z 1157.3,A -85,B 0,C 180,E1 11992.259,E2 11992.259} C_VEL
LIN {X 0,Y 260.206,Z 1167.557,A -85,B 0,C 180,E1 11989.061,E2 11989.061} C_VEL
LIN {X 0,Y 256.943,Z 1176.236,A -85,B 0,C 180,E1 11985.572,E2 11985.572} C_VEL
LIN {X 0,Y 254.412,Z 1182.875,A -85,B 0,C 180,E1 11982.019,E2 11982.019} C_VEL
LIN {X 0,Y 252.497,Z 1187.984,A -85,B 0,C 180,E1 11978.193,E2 11978.193} C_VEL
LIN {X 0,Y 251.28,Z 1191.488,A -85,B 0,C 180,E1 11974.104,E2 11974.104} C_VEL
LIN {X 0,Y 250.816,Z 1193.098,A -85,B 0,C 180,E1 11970.225,E2 11970.225} C_VEL
LIN {X 0,Y 250.968,Z 1192.995,A -85,B 0,C 180,E1 11966.113,E2 11966.113} C_VEL
LIN {X 0,Y 251.83,Z 1191.099,A -85,B 0,C 180,E1 11962.009,E2 11962.009} C_VEL
LIN {X 0,Y 253.4,Z 1187.557,A -85,B 0,C 180,E1 11958.122,E2 11958.122} C_VEL
LIN {X 0,Y 255.709,Z 1182.253,A -85,B 0,C 180,E1 11954.344,E2 11954.344} C_VEL
LIN {X 0,Y 258.659,Z 1175.363,A -85,B 0,C 180,E1 11950.814,E2 11950.814} C_VEL
LIN {X 0,Y 262.36,Z 1166.441,A -85,B 0,C 180,E1 11947.358,E2 11947.358} C_VEL
LIN {X 0,Y 266.386,Z 1156.117,A -85,B 0,C 180,E1 11944.271,E2 11944.271} C_VEL
LIN {X 0,Y 270.544,Z 1144.375,A -85,B 0,C 180,E1 11941.523,E2 11941.523} C_VEL
LIN {X 0,Y 274.656,Z 1131.41,A -85,B 0,C 180,E1 11939.113,E2 11939.113} C_VEL
LIN {X 0,Y 278.514,Z 1117.448,A -85,B 0,C 180,E1 11937.048,E2 11937.048} C_VEL
LIN {X 0,Y 281.954,Z 1102.394,A -85,B 0,C 180,E1 11935.304,E2 11935.304} C_VEL
LIN {X 0,Y 284.863,Z 1086.234,A -85,B 0,C 180,E1 11933.862,E2 11933.862} C_VEL
LIN {X 0,Y 287.102,Z 1069.155,A -85,B 0,C 180,E1 11932.73,E2 11932.73} C_VEL
LIN {X 0,Y 288.461,Z 1051.911,A -85,B 0,C 180,E1 11931.947,E2 11931.947} C_VEL
LIN {X 0,Y 288.983,Z 1040.032,A -85,B 0,C 180,E1 11931.571,E2 11931.571} C_VEL
LIN {X 0,Y 290.81,Z 1040.701,A -85,B 0,C 180,E1 11931.259,E2 11931.259} C_VEL
LIN {X 0,Y 293.221,Z 1039.807,A -85,B 0,C 180,E1 11931.031,E2 11931.031} C_VEL
LIN {X 0,Y 296.263,Z 1036.752,A -85,B 0,C 180,E1 11930.919,E2 11930.919} C_VEL
LIN {X 0,Y 299.658,Z 1031.41,A -85,B 0,C 180,E1 11930.967,E2 11930.967} C_VEL
LIN {X 0,Y 303.787,Z 1028.738,A -85,B 0,C 180,E1 11930.668,E2 11930.668} C_VEL
LIN {X 0,Y 307.567,Z 1024.605,A -85,B 0,C 180,E1 11930.544,E2 11930.544} C_VEL
LIN {X 0,Y 311.69,Z 1017.548,A -85,B 0,C 180,E1 11930.564,E2 11930.564} C_VEL
LIN {X 0,Y 312.826,Z 1016.695,A -85,B 0,C 180,E1 11930.484,E2 11930.484} C_VEL
LIN {X 0,Y 308.004,Z 1040.7,A -85,B 0,C 180,E1 11929.048,E2 11929.048} C_VEL
LIN {X 0,Y 302.62,Z 1063.161,A -85,B 0,C 180,E1 11927.361,E2 11927.361} C_VEL
LIN {X 0,Y 296.643,Z 1084.984,A -85,B 0,C 180,E1 11925.334,E2 11925.334} C_VEL
LIN {X 0,Y 290.068,Z 1106.329,A -85,B 0,C 180,E1 11922.907,E2 11922.907} C_VEL
LIN {X 0,Y 283.492,Z 1125.949,A -85,B 0,C 180,E1 11920.2,E2 11920.2} C_VEL
LIN {X 0,Y 281.958,Z 1130.434,A -85,B 0,C 180,E1 11919.51,E2 11919.51} C_VEL
LIN {X 0,Y 278.974,Z 1136.279,A -85,B 0,C 180,E1 11918.64,E2 11918.64} C_VEL
LIN {X 0,Y 267.821,Z 1151.059,A -85,B 0,C 180,E1 11916.451,E2 11916.451} C_VEL
LIN {X 0,Y 265.38,Z 1155.622,A -85,B 0,C 180,E1 11915.568,E2 11915.568} C_VEL
LIN {X 0,Y 258.975,Z 1172.544,A -85,B 0,C 180,E1 11911.675,E2 11911.675} C_VEL
LIN {X 0,Y 253.397,Z 1187.56,A -85,B 0,C 180,E1 11907.495,E2 11907.495} C_VEL
LIN {X 0,Y 248.891,Z 1200.454,A -85,B 0,C 180,E1 11903.185,E2 11903.185} C_VEL
LIN {X 0,Y 245.131,Z 1212.469,A -85,B 0,C 180,E1 11898.306,E2 11898.306} C_VEL
LIN {X 0,Y 242.622,Z 1222.272,A -85,B 0,C 180,E1 11893.434,E2 11893.434} C_VEL
LIN {X 0,Y 241.11,Z 1230.596,A -85,B 0,C 180,E1 11888.346,E2 11888.346} C_VEL
LIN {X 0,Y 240.5,Z 1236.883,A -85,B 0,C 180,E1 11883.576,E2 11883.576} C_VEL
LIN {X 0,Y 240.391,Z 1241.679,A -85,B 0,C 180,E1 11878.808,E2 11878.808} C_VEL
LIN {X 0,Y 240.643,Z 1245.493,A -85,B 0,C 180,E1 11873.798,E2 11873.798} C_VEL
LIN {X 0,Y 241.516,Z 1248.026,A -85,B 0,C 180,E1 11868.538,E2 11868.538} C_VEL
LIN {X 0,Y 243.975,Z 1249.458,A -85,B 0,C 180,E1 11862.345,E2 11862.345} C_VEL
LIN {X 0,Y 248.765,Z 1249.183,A -85,B 0,C 180,E1 11856.048,E2 11856.048} C_VEL
LIN {X 0,Y 256.488,Z 1247.112,A -85,B 0,C 180,E1 11849.808,E2 11849.808} C_VEL
LIN {X 0,Y 267.946,Z 1242.979,A -85,B 0,C 180,E1 11843.606,E2 11843.606} C_VEL
LIN {X 0,Y 282.07,Z 1237.209,A -85,B 0,C 180,E1 11838.208,E2 11838.208} C_VEL
LIN {X 0,Y 293.361,Z 1232.322,A -85,B 0,C 180,E1 11834.876,E2 11834.876} C_VEL
LIN {X 0,Y 275.503,Z 1242.87,A -85,B 0,C 180,E1 11829.973,E2 11829.973} C_VEL
LIN {X 0,Y 261.067,Z 1252.646,A -85,B 0,C 180,E1 11824.179,E2 11824.179} C_VEL
LIN {X 0,Y 250.976,Z 1260.509,A -85,B 0,C 180,E1 11818.045,E2 11818.045} C_VEL
LIN {X 0,Y 244.66,Z 1266.223,A -85,B 0,C 180,E1 11811.836,E2 11811.836} C_VEL
LIN {X 0,Y 241.434,Z 1269.727,A -85,B 0,C 180,E1 11805.866,E2 11805.866} C_VEL
LIN {X 0,Y 240.388,Z 1271.202,A -85,B 0,C 180,E1 11800.549,E2 11800.549} C_VEL
LIN {X 0,Y 240.477,Z 1271.059,A -85,B 0,C 180,E1 11795.73,E2 11795.73} C_VEL
LIN {X 0,Y 240.871,Z 1269.555,A -85,B 0,C 180,E1 11791.43,E2 11791.43} C_VEL
LIN {X 0,Y 241.034,Z 1267.061,A -85,B 0,C 180,E1 11787.626,E2 11787.626} C_VEL
LIN {X 0,Y 240.973,Z 1263.097,A -85,B 0,C 180,E1 11783.571,E2 11783.571} C_VEL
LIN {X 0,Y 241.005,Z 1257.339,A -85,B 0,C 180,E1 11779.243,E2 11779.243} C_VEL
LIN {X 0,Y 241.575,Z 1249.515,A -85,B 0,C 180,E1 11774.643,E2 11774.643} C_VEL
LIN {X 0,Y 243.077,Z 1239.286,A -85,B 0,C 180,E1 11769.789,E2 11769.789} C_VEL
LIN {X 0,Y 245.718,Z 1226.996,A -85,B 0,C 180,E1 11764.967,E2 11764.967} C_VEL
LIN {X 0,Y 249.645,Z 1212.403,A -85,B 0,C 180,E1 11760.225,E2 11760.225} C_VEL
LIN {X 0,Y 254.927,Z 1195.462,A -85,B 0,C 180,E1 11755.616,E2 11755.616} C_VEL
LIN {X 0,Y 261.805,Z 1175.396,A -85,B 0,C 180,E1 11751.083,E2 11751.083} C_VEL
LIN {X 0,Y 270.149,Z 1152.272,A -85,B 0,C 180,E1 11746.79,E2 11746.79} C_VEL
LIN {X 0,Y 279.168,Z 1127.696,A -85,B 0,C 180,E1 11743.063,E2 11743.063} C_VEL
LIN {X 0,Y 289.436,Z 1099.659,A -85,B 0,C 180,E1 11739.617,E2 11739.617} C_VEL
LIN {X 0,Y 299.348,Z 1072.529,A -85,B 0,C 180,E1 11736.877,E2 11736.877} C_VEL
LIN {X 0,Y 309.134,Z 1044.732,A -85,B 0,C 180,E1 11734.602,E2 11734.602} C_VEL
LIN {X 0,Y 318.582,Z 1016.59,A -85,B 0,C 180,E1 11732.746,E2 11732.746} C_VEL
LIN {X 0,Y 322.836,Z 1003.06,A -85,B 0,C 180,E1 11731.98,E2 11731.98} C_VEL
LIN {X 0,Y 319.603,Z 979.554,A -85,B 0,C 180,E1 11729.316,E2 11729.316} C_VEL
LIN {X 0,Y 317.468,Z 954.335,A -85,B 0,C 180,E1 11726.769,E2 11726.769} C_VEL
LIN {X 0,Y 316.292,Z 927.23,A -85,B 0,C 180,E1 11724.409,E2 11724.409} C_VEL
LIN {X 0,Y 316.195,Z 898.86,A -85,B 0,C 180,E1 11722.313,E2 11722.313} C_VEL
LIN {X 0,Y 316.991,Z 875.051,A -85,B 0,C 180,E1 11720.688,E2 11720.688} C_VEL
LIN {X 0,Y 327.763,Z 842.156,A -85,B 0,C 180,E1 11716.482,E2 11716.482} C_VEL
LIN {X 0,Y 327.986,Z 840.923,A -85,B 0,C 180,E1 11716.288,E2 11716.288} C_VEL
LIN {X 0,Y 322.916,Z 825.77,A -85,B 0,C 180,E1 11712.337,E2 11712.337} C_VEL
LIN {X 0,Y 317.224,Z 809.912,A -85,B 0,C 180,E1 11707.79,E2 11707.79} C_VEL
LIN {X 0,Y 312.249,Z 796.878,A -85,B 0,C 180,E1 11703.672,E2 11703.672} C_VEL
LIN {X 0,Y 307.648,Z 785.182,A -85,B 0,C 180,E1 11699.628,E2 11699.628} C_VEL
LIN {X 0,Y 302.946,Z 773.746,A -85,B 0,C 180,E1 11695.267,E2 11695.267} C_VEL
LIN {X 0,Y 298.584,Z 763.559,A -85,B 0,C 180,E1 11690.944,E2 11690.944} C_VEL
LIN {X 0,Y 294.429,Z 753.896,A -85,B 0,C 180,E1 11686.448,E2 11686.448} C_VEL
LIN {X 0,Y 290.398,Z 745.144,A -85,B 0,C 180,E1 11681.852,E2 11681.852} C_VEL
LIN {X 0,Y 287.62,Z 739.196,A -85,B 0,C 180,E1 11678.377,E2 11678.377} C_VEL
LIN {X 0,Y 284.802,Z 732.942,A -85,B 0,C 180,E1 11674.416,E2 11674.416} C_VEL
LIN {X 0,Y 283.651,Z 730.648,A -85,B 0,C 180,E1 11672.725,E2 11672.725} C_VEL
LIN {X 0,Y 289.718,Z 732.18,A -85,B 0,C 180,E1 11670.37,E2 11670.37} C_VEL
LIN {X 0,Y 294.625,Z 744.942,A -85,B 0,C 180,E1 11666.88,E2 11666.88} C_VEL
LIN {X 0,Y 298.887,Z 758.435,A -85,B 0,C 180,E1 11663.691,E2 11663.691} C_VEL
LIN {X 0,Y 302.718,Z 772.925,A -85,B 0,C 180,E1 11660.763,E2 11660.763} C_VEL
LIN {X 0,Y 303.142,Z 775.197,A -85,B 0,C 180,E1 11660.365,E2 11660.365} C_VEL
LIN {X 0,Y 295.723,Z 821.444,A -85,B 0,C 180,E1 11655.926,E2 11655.926} C_VEL
LIN {X 0,Y 288.26,Z 871.951,A -85,B 0,C 180,E1 11651.092,E2 11651.092} C_VEL
LIN {X 0,Y 287.203,Z 880.733,A -85,B 0,C 180,E1 11650.3,E2 11650.3} C_VEL
LIN {X 0,Y 287.366,Z 887.176,A -85,B 0,C 180,E1 11650.061,E2 11650.061} C_VEL
LIN {X 0,Y 279.479,Z 1035.239,A -85,B 0,C 180,E1 11646.601,E2 11646.601} C_VEL
LIN {X 0,Y 278.602,Z 1056.6,A -85,B 0,C 180,E1 11645.926,E2 11645.926} C_VEL
LIN {X 0,Y 276.999,Z 1074.379,A -85,B 0,C 180,E1 11645.004,E2 11645.004} C_VEL
LIN {X 0,Y 274.754,Z 1090.39,A -85,B 0,C 180,E1 11643.831,E2 11643.831} C_VEL
LIN {X 0,Y 271.683,Z 1106.502,A -85,B 0,C 180,E1 11642.249,E2 11642.249} C_VEL
LIN {X 0,Y 267.956,Z 1122.204,A -85,B 0,C 180,E1 11640.245,E2 11640.245} C_VEL
LIN {X 0,Y 264.07,Z 1136.026,A -85,B 0,C 180,E1 11637.999,E2 11637.999} C_VEL
LIN {X 0,Y 260.148,Z 1148.226,A -85,B 0,C 180,E1 11635.494,E2 11635.494} C_VEL
LIN {X 0,Y 256.039,Z 1159.798,A -85,B 0,C 180,E1 11632.498,E2 11632.498} C_VEL
LIN {X 0,Y 252.25,Z 1169.783,A -85,B 0,C 180,E1 11629.205,E2 11629.205} C_VEL
LIN {X 0,Y 249.115,Z 1177.703,A -85,B 0,C 180,E1 11625.836,E2 11625.836} C_VEL
LIN {X 0,Y 246.482,Z 1184.251,A -85,B 0,C 180,E1 11622.134,E2 11622.134} C_VEL
LIN {X 0,Y 244.456,Z 1189.444,A -85,B 0,C 180,E1 11617.991,E2 11617.991} C_VEL
LIN {X 0,Y 243.313,Z 1192.607,A -85,B 0,C 180,E1 11614.003,E2 11614.003} C_VEL
LIN {X 0,Y 242.854,Z 1194.11,A -85,B 0,C 180,E1 11609.761,E2 11609.761} C_VEL
LIN {X 0,Y 243.102,Z 1193.815,A -85,B 0,C 180,E1 11605.515,E2 11605.515} C_VEL
LIN {X 0,Y 244.11,Z 1191.737,A -85,B 0,C 180,E1 11601.28,E2 11601.28} C_VEL
LIN {X 0,Y 245.841,Z 1187.998,A -85,B 0,C 180,E1 11597.31,E2 11597.31} C_VEL
LIN {X 0,Y 248.394,Z 1182.397,A -85,B 0,C 180,E1 11593.39,E2 11593.39} C_VEL
LIN {X 0,Y 251.77,Z 1174.903,A -85,B 0,C 180,E1 11589.597,E2 11589.597} C_VEL
LIN {X 0,Y 255.571,Z 1166.08,A -85,B 0,C 180,E1 11586.233,E2 11586.233} C_VEL
LIN {X 0,Y 259.652,Z 1155.892,A -85,B 0,C 180,E1 11583.218,E2 11583.218} C_VEL
LIN {X 0,Y 263.917,Z 1144.26,A -85,B 0,C 180,E1 11580.49,E2 11580.49} C_VEL
LIN {X 0,Y 268.234,Z 1131.079,A -85,B 0,C 180,E1 11578.037,E2 11578.037} C_VEL
LIN {X 0,Y 272.258,Z 1116.726,A -85,B 0,C 180,E1 11575.937,E2 11575.937} C_VEL
LIN {X 0,Y 275.846,Z 1101.231,A -85,B 0,C 180,E1 11574.165,E2 11574.165} C_VEL
LIN {X 0,Y 278.765,Z 1085.169,A -85,B 0,C 180,E1 11572.754,E2 11572.754} C_VEL
LIN {X 0,Y 280.954,Z 1068.308,A -85,B 0,C 180,E1 11571.663,E2 11571.663} C_VEL
LIN {X 0,Y 282.265,Z 1053.975,A -85,B 0,C 180,E1 11570.972,E2 11570.972} C_VEL
LIN {X 0,Y 284.022,Z 1054.467,A -85,B 0,C 180,E1 11570.675,E2 11570.675} C_VEL
LIN {X 0,Y 286.686,Z 1053.562,A -85,B 0,C 180,E1 11570.426,E2 11570.426} C_VEL
LIN {X 0,Y 289.744,Z 1050.887,A -85,B 0,C 180,E1 11570.323,E2 11570.323} C_VEL
LIN {X 0,Y 292.512,Z 1047.328,A -85,B 0,C 180,E1 11570.341,E2 11570.341} C_VEL
LIN {X 0,Y 296.63,Z 1045.03,A -85,B 0,C 180,E1 11570.045,E2 11570.045} C_VEL
LIN {X 0,Y 300.505,Z 1041.226,A -85,B 0,C 180,E1 11569.934,E2 11569.934} C_VEL
LIN {X 0,Y 301.511,Z 1039.963,A -85,B 0,C 180,E1 11569.932,E2 11569.932} C_VEL
LIN {X 0,Y 295.896,Z 1062.916,A -85,B 0,C 180,E1 11568.193,E2 11568.193} C_VEL
LIN {X 0,Y 289.44,Z 1085.9,A -85,B 0,C 180,E1 11566.02,E2 11566.02} C_VEL
LIN {X 0,Y 282.814,Z 1106.855,A -85,B 0,C 180,E1 11563.585,E2 11563.585} C_VEL
LIN {X 0,Y 275.986,Z 1126.729,A -85,B 0,C 180,E1 11560.779,E2 11560.779} C_VEL
LIN {X 0,Y 269.106,Z 1145.655,A -85,B 0,C 180,E1 11557.543,E2 11557.543} C_VEL
LIN {X 0,Y 265.38,Z 1155.622,A -85,B 0,C 180,E1 11555.568,E2 11555.568} C_VEL
LIN {X 0,Y 262.454,Z 1160.93,A -85,B 0,C 180,E1 11554.512,E2 11554.512} C_VEL
LIN {X 0,Y 251.445,Z 1174.22,A -85,B 0,C 180,E1 11551.743,E2 11551.743} C_VEL
LIN {X 0,Y 249.124,Z 1178.333,A -85,B 0,C 180,E1 11550.665,E2 11550.665} C_VEL
LIN {X 0,Y 243.521,Z 1193.35,A -85,B 0,C 180,E1 11546.062,E2 11546.062} C_VEL
LIN {X 0,Y 239.163,Z 1205.975,A -85,B 0,C 180,E1 11541.329,E2 11541.329} C_VEL
LIN {X 0,Y 235.989,Z 1216.657,A -85,B 0,C 180,E1 11536.492,E2 11536.492} C_VEL
LIN {X 0,Y 233.854,Z 1226.03,A -85,B 0,C 180,E1 11531.343,E2 11531.343} C_VEL
LIN {X 0,Y 232.782,Z 1233.29,A -85,B 0,C 180,E1 11526.412,E2 11526.412} C_VEL
LIN {X 0,Y 232.406,Z 1239.309,A -85,B 0,C 180,E1 11521.233,E2 11521.233} C_VEL
LIN {X 0,Y 232.462,Z 1243.772,A -85,B 0,C 180,E1 11516.301,E2 11516.301} C_VEL
LIN {X 0,Y 233.028,Z 1247.188,A -85,B 0,C 180,E1 11510.865,E2 11510.865} C_VEL
LIN {X 0,Y 234.791,Z 1249.568,A -85,B 0,C 180,E1 11504.69,E2 11504.69} C_VEL
LIN {X 0,Y 238.602,Z 1250.412,A -85,B 0,C 180,E1 11498.36,E2 11498.36} C_VEL
LIN {X 0,Y 245.429,Z 1249.54,A -85,B 0,C 180,E1 11491.797,E2 11491.797} C_VEL
LIN {X 0,Y 255.62,Z 1246.826,A -85,B 0,C 180,E1 11485.446,E2 11485.446} C_VEL
LIN {X 0,Y 269.175,Z 1242.298,A -85,B 0,C 180,E1 11479.6,E2 11479.6} C_VEL
LIN {X 0,Y 283.726,Z 1236.919,A -85,B 0,C 180,E1 11474.961,E2 11474.961} C_VEL
LIN {X 0,Y 265.727,Z 1246.771,A -85,B 0,C 180,E1 11469.771,E2 11469.771} C_VEL
LIN {X 0,Y 251.287,Z 1255.756,A -85,B 0,C 180,E1 11463.582,E2 11463.582} C_VEL
LIN {X 0,Y 241.512,Z 1262.671,A -85,B 0,C 180,E1 11457.095,E2 11457.095} C_VEL
LIN {X 0,Y 235.864,Z 1267.245,A -85,B 0,C 180,E1 11450.864,E2 11450.864} C_VEL
LIN {X 0,Y 233.123,Z 1269.814,A -85,B 0,C 180,E1 11444.916,E2 11444.916} C_VEL
LIN {X 0,Y 232.364,Z 1270.582,A -85,B 0,C 180,E1 11439.414,E2 11439.414} C_VEL
LIN {X 0,Y 232.625,Z 1269.819,A -85,B 0,C 180,E1 11434.688,E2 11434.688} C_VEL
LIN {X 0,Y 233.021,Z 1267.935,A -85,B 0,C 180,E1 11430.495,E2 11430.495} C_VEL
LIN {X 0,Y 233.11,Z 1264.993,A -85,B 0,C 180,E1 11426.561,E2 11426.561} C_VEL
LIN {X 0,Y 233.028,Z 1260.459,A -85,B 0,C 180,E1 11422.36,E2 11422.36} C_VEL
LIN {X 0,Y 233.195,Z 1253.738,A -85,B 0,C 180,E1 11417.624,E2 11417.624} C_VEL
LIN {X 0,Y 234.04,Z 1245.213,A -85,B 0,C 180,E1 11412.859,E2 11412.859} C_VEL
LIN {X 0,Y 235.982,Z 1234.179,A -85,B 0,C 180,E1 11407.849,E2 11407.849} C_VEL
LIN {X 0,Y 239.168,Z 1221.014,A -85,B 0,C 180,E1 11402.894,E2 11402.894} C_VEL
LIN {X 0,Y 243.719,Z 1205.527,A -85,B 0,C 180,E1 11398.05,E2 11398.05} C_VEL
LIN {X 0,Y 249.7,Z 1187.616,A -85,B 0,C 180,E1 11393.374,E2 11393.374} C_VEL
LIN {X 0,Y 257.323,Z 1166.4,A -85,B 0,C 180,E1 11388.809,E2 11388.809} C_VEL
LIN {X 0,Y 265.961,Z 1143.249,A -85,B 0,C 180,E1 11384.725,E2 11384.725} C_VEL
LIN {X 0,Y 275.593,Z 1117.685,A -85,B 0,C 180,E1 11381.049,E2 11381.049} C_VEL
LIN {X 0,Y 285.992,Z 1089.942,A -85,B 0,C 180,E1 11377.806,E2 11377.806} C_VEL
LIN {X 0,Y 296.084,Z 1062.57,A -85,B 0,C 180,E1 11375.196,E2 11375.196} C_VEL
LIN {X 0,Y 306.664,Z 1032.875,A -85,B 0,C 180,E1 11372.909,E2 11372.909} C_VEL
LIN {X 0,Y 316.033,Z 1004.459,A -85,B 0,C 180,E1 11371.151,E2 11371.151} C_VEL
LIN {X 0,Y 313.007,Z 979.87,A -85,B 0,C 180,E1 11368.319,E2 11368.319} C_VEL
LIN {X 0,Y 311.346,Z 956.385,A -85,B 0,C 180,E1 11365.898,E2 11365.898} C_VEL
LIN {X 0,Y 310.51,Z 928.56,A -85,B 0,C 180,E1 11363.41,E2 11363.41} C_VEL
LIN {X 0,Y 310.679,Z 900.967,A -85,B 0,C 180,E1 11361.326,E2 11361.326} C_VEL
LIN {X 0,Y 311.851,Z 872.666,A -85,B 0,C 180,E1 11359.357,E2 11359.357} C_VEL
LIN {X 0,Y 321.329,Z 844.443,A -85,B 0,C 180,E1 11355.707,E2 11355.707} C_VEL
LIN {X 0,Y 316.263,Z 829.266,A -85,B 0,C 180,E1 11351.674,E2 11351.674} C_VEL
LIN {X 0,Y 311.049,Z 814.539,A -85,B 0,C 180,E1 11347.388,E2 11347.388} C_VEL
LIN {X 0,Y 306.328,Z 802.003,A -85,B 0,C 180,E1 11343.368,E2 11343.368} C_VEL
LIN {X 0,Y 301.759,Z 790.221,A -85,B 0,C 180,E1 11339.241,E2 11339.241} C_VEL
LIN {X 0,Y 296.928,Z 778.245,A -85,B 0,C 180,E1 11334.59,E2 11334.59} C_VEL
LIN {X 0,Y 292.176,Z 767.052,A -85,B 0,C 180,E1 11329.749,E2 11329.749} C_VEL
LIN {X 0,Y 288.145,Z 757.962,A -85,B 0,C 180,E1 11325.326,E2 11325.326} C_VEL
LIN {X 0,Y 284.679,Z 750.212,A -85,B 0,C 180,E1 11321.147,E2 11321.147} C_VEL
LIN {X 0,Y 281.807,Z 743.562,A -85,B 0,C 180,E1 11317.248,E2 11317.248} C_VEL
LIN {X 0,Y 279.018,Z 737.89,A -85,B 0,C 180,E1 11313.388,E2 11313.388} C_VEL
LIN {X 0,Y 279.144,Z 737.816,A -85,B 0,C 180,E1 11313.171,E2 11313.171} C_VEL
LIN {X 0,Y 284.993,Z 739.052,A -85,B 0,C 180,E1 11310.812,E2 11310.812} C_VEL
LIN {X 0,Y 285.625,Z 739.401,A -85,B 0,C 180,E1 11310.538,E2 11310.538} C_VEL
LIN {X 0,Y 289.988,Z 751.417,A -85,B 0,C 180,E1 11307.225,E2 11307.225} C_VEL
LIN {X 0,Y 294.033,Z 764.884,A -85,B 0,C 180,E1 11304.026,E2 11304.026} C_VEL
LIN {X 0,Y 297.435,Z 778.326,A -85,B 0,C 180,E1 11301.297,E2 11301.297} C_VEL
LIN {X 0,Y 289.288,Z 827.598,A -85,B 0,C 180,E1 11296.534,E2 11296.534} C_VEL
LIN {X 0,Y 281.494,Z 878.539,A -85,B 0,C 180,E1 11291.62,E2 11291.62} C_VEL
LIN {X 0,Y 281.238,Z 881.998,A -85,B 0,C 180,E1 11291.346,E2 11291.346} C_VEL
LIN {X 0,Y 281.353,Z 888.132,A -85,B 0,C 180,E1 11291.116,E2 11291.116} C_VEL
LIN {X 0,Y 273.191,Z 1035.601,A -85,B 0,C 180,E1 11287.624,E2 11287.624} C_VEL
LIN {X 0,Y 272.252,Z 1057.427,A -85,B 0,C 180,E1 11286.925,E2 11286.925} C_VEL
LIN {X 0,Y 270.579,Z 1075.229,A -85,B 0,C 180,E1 11285.988,E2 11285.988} C_VEL
LIN {X 0,Y 268.204,Z 1091.509,A -85,B 0,C 180,E1 11284.774,E2 11284.774} C_VEL
LIN {X 0,Y 265.009,Z 1107.577,A -85,B 0,C 180,E1 11283.164,E2 11283.164} C_VEL
LIN {X 0,Y 261.136,Z 1123.258,A -85,B 0,C 180,E1 11281.122,E2 11281.122} C_VEL
LIN {X 0,Y 257.093,Z 1137.062,A -85,B 0,C 180,E1 11278.829,E2 11278.829} C_VEL
LIN {X 0,Y 252.769,Z 1149.905,A -85,B 0,C 180,E1 11276.109,E2 11276.109} C_VEL
LIN {X 0,Y 248.44,Z 1161.552,A -85,B 0,C 180,E1 11272.975,E2 11272.975} C_VEL
LIN {X 0,Y 244.528,Z 1171.382,A -85,B 0,C 180,E1 11269.587,E2 11269.587} C_VEL
LIN {X 0,Y 241.097,Z 1179.575,A -85,B 0,C 180,E1 11265.882,E2 11265.882} C_VEL
LIN {X 0,Y 238.322,Z 1186.193,A -85,B 0,C 180,E1 11261.86,E2 11261.86} C_VEL
LIN {X 0,Y 236.414,Z 1190.903,A -85,B 0,C 180,E1 11257.775,E2 11257.775} C_VEL
LIN {X 0,Y 235.299,Z 1193.815,A -85,B 0,C 180,E1 11253.651,E2 11253.651} C_VEL
LIN {X 0,Y 234.901,Z 1195.11,A -85,B 0,C 180,E1 11249.265,E2 11249.265} C_VEL
LIN {X 0,Y 235.258,Z 1194.637,A -85,B 0,C 180,E1 11244.876,E2 11244.876} C_VEL
LIN {X 0,Y 236.336,Z 1192.517,A -85,B 0,C 180,E1 11240.745,E2 11240.745} C_VEL
LIN {X 0,Y 238.212,Z 1188.638,A -85,B 0,C 180,E1 11236.649,E2 11236.649} C_VEL
LIN {X 0,Y 240.961,Z 1182.93,A -85,B 0,C 180,E1 11232.613,E2 11232.613} C_VEL
LIN {X 0,Y 244.39,Z 1175.676,A -85,B 0,C 180,E1 11228.882,E2 11228.882} C_VEL
LIN {X 0,Y 248.304,Z 1166.977,A -85,B 0,C 180,E1 11225.492,E2 11225.492} C_VEL
LIN {X 0,Y 252.57,Z 1156.776,A -85,B 0,C 180,E1 11222.404,E2 11222.404} C_VEL
LIN {X 0,Y 257.02,Z 1145.13,A -85,B 0,C 180,E1 11219.616,E2 11219.616} C_VEL
LIN {X 0,Y 261.516,Z 1131.93,A -85,B 0,C 180,E1 11217.114,E2 11217.114} C_VEL
LIN {X 0,Y 265.701,Z 1117.542,A -85,B 0,C 180,E1 11214.975,E2 11214.975} C_VEL
LIN {X 0,Y 269.431,Z 1102.012,A -85,B 0,C 180,E1 11213.174,E2 11213.174} C_VEL
LIN {X 0,Y 272.405,Z 1086.25,A -85,B 0,C 180,E1 11211.768,E2 11211.768} C_VEL
LIN {X 0,Y 274.694,Z 1069.395,A -85,B 0,C 180,E1 11210.656,E2 11210.656} C_VEL
LIN {X 0,Y 275.174,Z 1066.008,A -85,B 0,C 180,E1 11210.443,E2 11210.443} C_VEL
LIN {X 0,Y 277.411,Z 1066.475,A -85,B 0,C 180,E1 11210.088,E2 11210.088} C_VEL
LIN {X 0,Y 280.607,Z 1065.239,A -85,B 0,C 180,E1 11209.834,E2 11209.834} C_VEL
LIN {X 0,Y 284.221,Z 1061.883,A -85,B 0,C 180,E1 11209.766,E2 11209.766} C_VEL
LIN {X 0,Y 284.832,Z 1061.25,A -85,B 0,C 180,E1 11209.762,E2 11209.762} C_VEL
LIN {X 0,Y 289.104,Z 1059.359,A -85,B 0,C 180,E1 11209.44,E2 11209.44} C_VEL
LIN {X 0,Y 290.223,Z 1058.603,A -85,B 0,C 180,E1 11209.385,E2 11209.385} C_VEL
LIN {X 0,Y 283.807,Z 1081.512,A -85,B 0,C 180,E1 11207.272,E2 11207.272} C_VEL
LIN {X 0,Y 276.848,Z 1103.498,A -85,B 0,C 180,E1 11204.772,E2 11204.772} C_VEL
LIN {X 0,Y 269.857,Z 1123.663,A -85,B 0,C 180,E1 11201.975,E2 11201.975} C_VEL
LIN {X 0,Y 263.016,Z 1142.257,A -85,B 0,C 180,E1 11198.849,E2 11198.849} C_VEL
LIN {X 0,Y 256.266,Z 1159.864,A -85,B 0,C 180,E1 11195.272,E2 11195.272} C_VEL
LIN {X 0,Y 250.047,Z 1175.9,A -85,B 0,C 180,E1 11191.322,E2 11191.322} C_VEL
LIN {X 0,Y 249.124,Z 1178.333,A -85,B 0,C 180,E1 11190.665,E2 11190.665} C_VEL
LIN {X 0,Y 246.367,Z 1182.998,A -85,B 0,C 180,E1 11189.377,E2 11189.377} C_VEL
LIN {X 0,Y 235.926,Z 1194.672,A -85,B 0,C 180,E1 11185.947,E2 11185.947} C_VEL
LIN {X 0,Y 233.894,Z 1198.218,A -85,B 0,C 180,E1 11184.67,E2 11184.67} C_VEL
LIN {X 0,Y 229.769,Z 1210.571,A -85,B 0,C 180,E1 11179.578,E2 11179.578} C_VEL
LIN {X 0,Y 226.893,Z 1221.1,A -85,B 0,C 180,E1 11174.287,E2 11174.287} C_VEL
LIN {X 0,Y 225.218,Z 1229.744,A -85,B 0,C 180,E1 11168.939,E2 11168.939} C_VEL
LIN {X 0,Y 224.501,Z 1236.641,A -85,B 0,C 180,E1 11163.575,E2 11163.575} C_VEL
LIN {X 0,Y 224.396,Z 1241.881,A -85,B 0,C 180,E1 11158.468,E2 11158.468} C_VEL
LIN {X 0,Y 224.679,Z 1245.753,A -85,B 0,C 180,E1 11153.356,E2 11153.356} C_VEL
LIN {X 0,Y 225.711,Z 1248.836,A -85,B 0,C 180,E1 11147.723,E2 11147.723} C_VEL
LIN {X 0,Y 228.589,Z 1250.834,A -85,B 0,C 180,E1 11141.114,E2 11141.114} C_VEL
LIN {X 0,Y 234.352,Z 1251.204,A -85,B 0,C 180,E1 11134.198,E2 11134.198} C_VEL
LIN {X 0,Y 243.903,Z 1249.725,A -85,B 0,C 180,E1 11127.239,E2 11127.239} C_VEL
LIN {X 0,Y 257.42,Z 1246.235,A -85,B 0,C 180,E1 11120.718,E2 11120.718} C_VEL
LIN {X 0,Y 274.072,Z 1241.054,A -85,B 0,C 180,E1 11115.057,E2 11115.057} C_VEL
LIN {X 0,Y 255.95,Z 1250.203,A -85,B 0,C 180,E1 11109.555,E2 11109.555} C_VEL
LIN {X 0,Y 241.382,Z 1258.448,A -85,B 0,C 180,E1 11102.867,E2 11102.867} C_VEL
LIN {X 0,Y 232.103,Z 1264.339,A -85,B 0,C 180,E1 11096.07,E2 11096.07} C_VEL
LIN {X 0,Y 226.942,Z 1267.999,A -85,B 0,C 180,E1 11089.46,E2 11089.46} C_VEL
LIN {X 0,Y 224.782,Z 1269.629,A -85,B 0,C 180,E1 11083.378,E2 11083.378} C_VEL
LIN {X 0,Y 224.445,Z 1269.549,A -85,B 0,C 180,E1 11077.684,E2 11077.684} C_VEL
LIN {X 0,Y 224.863,Z 1268.123,A -85,B 0,C 180,E1 11073.062,E2 11073.062} C_VEL
LIN {X 0,Y 225.184,Z 1265.742,A -85,B 0,C 180,E1 11068.986,E2 11068.986} C_VEL
LIN {X 0,Y 225.174,Z 1262.146,A -85,B 0,C 180,E1 11064.908,E2 11064.908} C_VEL
LIN {X 0,Y 225.118,Z 1256.564,A -85,B 0,C 180,E1 11060.287,E2 11060.287} C_VEL
LIN {X 0,Y 225.551,Z 1248.939,A -85,B 0,C 180,E1 11055.367,E2 11055.367} C_VEL
LIN {X 0,Y 226.953,Z 1238.895,A -85,B 0,C 180,E1 11050.173,E2 11050.173} C_VEL
LIN {X 0,Y 229.645,Z 1226.456,A -85,B 0,C 180,E1 11044.911,E2 11044.911} C_VEL
LIN {X 0,Y 233.575,Z 1212.337,A -85,B 0,C 180,E1 11039.948,E2 11039.948} C_VEL
LIN {X 0,Y 239.029,Z 1195.534,A -85,B 0,C 180,E1 11035.039,E2 11035.039} C_VEL
